Yaskawa INFORM job: DEMO_ROOF_SIDE_0625_3PAINT_41.JBI

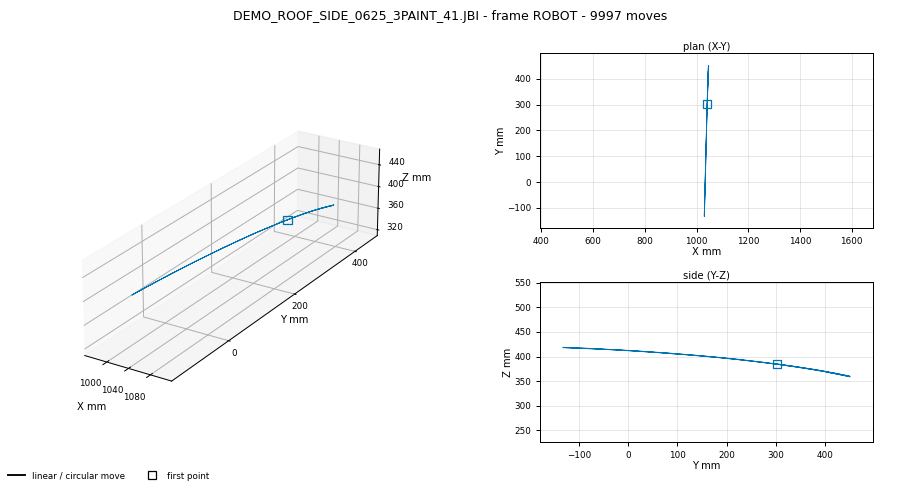
[picture p0: tool path of DEMO_ROOF_SIDE_0625_3PAINT_41.JBI in frame ROBOT, 9997 of 9997 moves have a stored position in this frame; points joined in program order, loops and branches not executed]
/JOB
//NAME DEMO_ROOF_SIDE_0625_3PAINT41
//POS
///NPOS 9997,0,0,0,0,0
///TOOL 0
///USER 0
///POSTYPE ROBOT
///RECTAN
///RCONF 1,0,0,0,0,0,0,0,0,0,0,0,0,0,0,0,0,0,0,0,0,0,0,0
C00000=1041.945,303.509,384.970,171.969,41.641,157.984
C00001=1041.951,303.756,384.937,171.973,41.643,157.985
C00002=1041.958,304.004,384.903,171.977,41.645,157.986
C00003=1041.965,304.251,384.871,171.981,41.648,157.987
C00004=1041.972,304.500,384.838,171.985,41.651,157.987
C00005=1041.979,304.747,384.804,171.988,41.653,157.988
C00006=1041.988,305.081,384.760,171.994,41.656,157.989
C00007=1041.997,305.416,384.715,171.999,41.659,157.990
C00008=1042.007,305.750,384.670,172.004,41.662,157.991
C00009=1042.016,306.084,384.626,172.010,41.665,157.992
C00010=1042.023,306.332,384.592,172.014,41.668,157.993
C00011=1042.030,306.580,384.559,172.018,41.670,157.994
C00012=1042.037,306.827,384.525,172.022,41.672,157.994
C00013=1042.044,307.075,384.491,172.026,41.675,157.995
C00014=1042.050,307.322,384.459,172.030,41.677,157.996
C00015=1042.057,307.570,384.425,172.034,41.680,157.997
C00016=1042.065,307.818,384.392,172.037,41.682,157.998
C00017=1042.072,308.065,384.359,172.041,41.685,157.998
C00018=1042.079,308.313,384.325,172.045,41.687,157.999
C00019=1042.086,308.561,384.292,172.049,41.689,158.000
C00020=1042.092,308.808,384.258,172.053,41.692,158.001
C00021=1042.100,309.056,384.225,172.057,41.694,158.001
C00022=1042.107,309.304,384.192,172.061,41.696,158.002
C00023=1042.114,309.551,384.159,172.065,41.699,158.003
C00024=1042.121,309.798,384.125,172.069,41.702,158.004
C00025=1042.128,310.046,384.091,172.073,41.703,158.005
C00026=1042.135,310.294,384.058,172.077,41.706,158.005
C00027=1042.142,310.541,384.024,172.081,41.709,158.006
C00028=1042.149,310.789,383.991,172.085,41.711,158.007
C00029=1042.156,311.037,383.957,172.089,41.713,158.008
C00030=1042.163,311.284,383.923,172.093,41.716,158.009
C00031=1042.170,311.531,383.890,172.097,41.718,158.009
C00032=1042.178,311.779,383.857,172.101,41.721,158.010
C00033=1042.185,312.027,383.823,172.106,41.723,158.011
C00034=1042.192,312.275,383.789,172.110,41.725,158.012
C00035=1042.198,312.523,383.755,172.114,41.728,158.013
C00036=1042.205,312.770,383.722,172.118,41.730,158.013
C00037=1042.212,313.017,383.688,172.122,41.733,158.014
C00038=1042.219,313.265,383.653,172.125,41.736,158.015
C00039=1042.226,313.512,383.619,172.130,41.739,158.016
C00040=1042.232,313.760,383.585,172.134,41.741,158.017
C00041=1042.239,314.007,383.551,172.138,41.744,158.018
C00042=1042.246,314.255,383.516,172.142,41.746,158.018
C00043=1042.253,314.503,383.483,172.146,41.749,158.019
C00044=1042.259,314.750,383.449,172.150,41.752,158.020
C00045=1042.266,314.997,383.414,172.154,41.754,158.021
C00046=1042.273,315.245,383.380,172.158,41.757,158.022
C00047=1042.280,315.493,383.346,172.162,41.759,158.023
C00048=1042.286,315.741,383.311,172.166,41.762,158.024
C00049=1042.294,315.988,383.277,172.170,41.765,158.024
C00050=1042.300,316.235,383.243,172.175,41.767,158.025
C00051=1042.307,316.483,383.209,172.179,41.770,158.026
C00052=1042.314,316.730,383.174,172.183,41.773,158.027
C00053=1042.321,316.978,383.140,172.187,41.775,158.028
C00054=1042.328,317.226,383.106,172.191,41.778,158.029
C00055=1042.335,317.473,383.071,172.195,41.781,158.029
C00056=1042.342,317.721,383.037,172.200,41.783,158.030
C00057=1042.349,317.968,383.002,172.204,41.786,158.031
C00058=1042.356,318.216,382.968,172.208,41.789,158.032
C00059=1042.362,318.463,382.934,172.212,41.792,158.033
C00060=1042.369,318.710,382.900,172.216,41.794,158.034
C00061=1042.376,318.958,382.865,172.221,41.797,158.035
C00062=1042.386,319.297,382.818,172.227,41.800,158.036
C00063=1042.395,319.636,382.771,172.232,41.804,158.037
C00064=1042.405,319.975,382.724,172.239,41.808,158.038
C00065=1042.415,320.314,382.676,172.244,41.811,158.039
C00066=1042.422,320.562,382.641,172.249,41.814,158.040
C00067=1042.429,320.809,382.607,172.253,41.817,158.041
C00068=1042.435,321.057,382.572,172.257,41.820,158.042
C00069=1042.443,321.304,382.538,172.261,41.822,158.043
C00070=1042.450,321.551,382.502,172.266,41.825,158.044
C00071=1042.457,321.799,382.469,172.270,41.828,158.045
C00072=1042.464,322.046,382.433,172.274,41.831,158.046
C00073=1042.470,322.294,382.398,172.278,41.833,158.047
C00074=1042.478,322.541,382.365,172.283,41.836,158.047
C00075=1042.485,322.789,382.329,172.287,41.839,158.048
C00076=1042.493,323.036,382.294,172.291,41.841,158.049
C00077=1042.499,323.284,382.259,172.296,41.844,158.050
C00078=1042.507,323.531,382.226,172.300,41.847,158.051
C00079=1042.513,323.779,382.190,172.304,41.850,158.052
C00080=1042.521,324.026,382.156,172.310,41.853,158.053
C00081=1042.528,324.273,382.121,172.313,41.855,158.054
C00082=1042.535,324.521,382.085,172.318,41.858,158.055
C00083=1042.542,324.768,382.051,172.323,41.861,158.056
C00084=1042.549,325.016,382.016,172.327,41.864,158.057
C00085=1042.556,325.263,381.982,172.331,41.866,158.057
C00086=1042.564,325.511,381.946,172.336,41.869,158.058
C00087=1042.571,325.759,381.912,172.340,41.872,158.059
C00088=1042.578,326.006,381.877,172.344,41.875,158.060
C00089=1042.585,326.253,381.841,172.349,41.877,158.061
C00090=1042.593,326.501,381.807,172.353,41.881,158.062
C00091=1042.600,326.748,381.771,172.357,41.883,158.063
C00092=1042.607,326.995,381.737,172.362,41.886,158.064
C00093=1042.615,327.244,381.701,172.366,41.889,158.065
C00094=1042.621,327.491,381.666,172.371,41.892,158.066
C00095=1042.629,327.738,381.632,172.375,41.894,158.067
C00096=1042.636,327.986,381.596,172.380,41.897,158.068
C00097=1042.644,328.233,381.562,172.385,41.900,158.069
C00098=1042.651,328.480,381.526,172.389,41.903,158.069
C00099=1042.658,328.728,381.490,172.394,41.906,158.070
C00100=1042.666,328.975,381.456,172.398,41.909,158.071
C00101=1042.672,329.222,381.421,172.402,41.911,158.072
C00102=1042.680,329.470,381.385,172.407,41.914,158.073
C00103=1042.687,329.717,381.349,172.411,41.918,158.074
C00104=1042.694,329.964,381.314,172.417,41.921,158.075
C00105=1042.701,330.213,381.279,172.421,41.924,158.076
C00106=1042.708,330.459,381.243,172.426,41.926,158.077
C00107=1042.715,330.707,381.208,172.430,41.929,158.078
C00108=1042.722,330.955,381.172,172.434,41.932,158.079
C00109=1042.729,331.201,381.136,172.439,41.935,158.080
C00110=1042.737,331.449,381.101,172.443,41.938,158.081
C00111=1042.744,331.696,381.065,172.449,41.941,158.082
C00112=1042.751,331.944,381.030,172.453,41.945,158.083
C00113=1042.758,332.191,380.994,172.458,41.948,158.084
C00114=1042.765,332.438,380.958,172.462,41.951,158.085
C00115=1042.773,332.686,380.922,172.467,41.954,158.086
C00116=1042.779,332.933,380.887,172.471,41.957,158.087
C00117=1042.787,333.181,380.851,172.476,41.960,158.088
C00118=1042.797,333.514,380.803,172.482,41.964,158.089
C00119=1042.807,333.849,380.754,172.489,41.968,158.091
C00120=1042.816,334.183,380.706,172.495,41.972,158.092
C00121=1042.826,334.517,380.658,172.501,41.976,158.093
C00122=1042.833,334.765,380.622,172.506,41.979,158.094
C00123=1042.841,335.012,380.586,172.510,41.982,158.095
C00124=1042.848,335.259,380.550,172.515,41.985,158.096
C00125=1042.856,335.507,380.515,172.520,41.988,158.097
C00126=1042.862,335.754,380.478,172.525,41.992,158.099
C00127=1042.870,336.001,380.442,172.529,41.995,158.100
C00128=1042.877,336.248,380.406,172.534,41.998,158.101
C00129=1042.884,336.496,380.369,172.540,42.001,158.102
C00130=1042.891,336.743,380.333,172.544,42.004,158.103
C00131=1042.898,336.990,380.297,172.549,42.007,158.104
C00132=1042.906,337.238,380.261,172.553,42.011,158.105
C00133=1042.912,337.485,380.224,172.559,42.014,158.106
C00134=1042.920,337.732,380.188,172.563,42.017,158.107
C00135=1042.928,337.979,380.152,172.568,42.020,158.108
C00136=1042.935,338.226,380.116,172.572,42.023,158.109
C00137=1042.942,338.474,380.079,172.577,42.026,158.110
C00138=1042.949,338.721,380.044,172.583,42.030,158.111
C00139=1042.956,338.968,380.007,172.587,42.033,158.112
C00140=1042.963,339.216,379.970,172.592,42.036,158.113
C00141=1042.970,339.463,379.935,172.597,42.040,158.114
C00142=1042.978,339.710,379.898,172.602,42.042,158.115
C00143=1042.985,339.958,379.862,172.607,42.046,158.116
C00144=1042.993,340.205,379.825,172.611,42.049,158.117
C00145=1043.000,340.451,379.789,172.617,42.053,158.119
C00146=1043.008,340.699,379.753,172.621,42.056,158.120
C00147=1043.015,340.947,379.716,172.626,42.059,158.121
C00148=1043.022,341.194,379.680,172.632,42.062,158.122
C00149=1043.030,341.440,379.643,172.636,42.065,158.123
C00150=1043.037,341.688,379.606,172.641,42.069,158.124
C00151=1043.044,341.935,379.570,172.646,42.072,158.125
C00152=1043.051,342.183,379.533,172.651,42.075,158.126
C00153=1043.059,342.430,379.496,172.656,42.079,158.127
C00154=1043.066,342.677,379.460,172.661,42.082,158.128
C00155=1043.074,342.924,379.423,172.666,42.086,158.129
C00156=1043.081,343.172,379.386,172.671,42.089,158.131
C00157=1043.089,343.418,379.349,172.676,42.092,158.132
C00158=1043.095,343.666,379.312,172.681,42.096,158.133
C00159=1043.103,343.912,379.276,172.686,42.099,158.134
C00160=1043.110,344.160,379.239,172.691,42.102,158.135
C00161=1043.118,344.407,379.202,172.696,42.106,158.136
C00162=1043.125,344.655,379.165,172.701,42.109,158.137
C00163=1043.132,344.902,379.128,172.706,42.112,158.138
C00164=1043.140,345.149,379.091,172.712,42.116,158.140
C00165=1043.147,345.396,379.054,172.716,42.120,158.141
C00166=1043.155,345.643,379.017,172.721,42.123,158.142
C00167=1043.162,345.890,378.979,172.727,42.127,158.143
C00168=1043.168,346.137,378.943,172.732,42.130,158.144
C00169=1043.176,346.384,378.906,172.736,42.133,158.145
C00170=1043.184,346.631,378.869,172.742,42.137,158.146
C00171=1043.191,346.878,378.831,172.747,42.140,158.148
C00172=1043.199,347.125,378.794,172.753,42.144,158.149
C00173=1043.206,347.373,378.757,172.757,42.147,158.150
C00174=1043.216,347.704,378.707,172.764,42.152,158.151
C00175=1043.226,348.034,378.658,172.771,42.157,158.153
C00176=1043.236,348.365,378.607,172.779,42.161,158.155
C00177=1043.246,348.695,378.558,172.785,42.166,158.156
C00178=1043.254,348.942,378.520,172.790,42.170,158.157
C00179=1043.261,349.189,378.483,172.795,42.173,158.159
C00180=1043.269,349.436,378.446,172.801,42.177,158.160
C00181=1043.277,349.683,378.408,172.806,42.180,158.161
C00182=1043.284,349.931,378.370,172.812,42.184,158.162
C00183=1043.291,350.178,378.333,172.817,42.188,158.163
C00184=1043.299,350.425,378.296,172.822,42.191,158.165
C00185=1043.306,350.672,378.258,172.827,42.195,158.166
C00186=1043.314,350.919,378.221,172.832,42.198,158.167
C00187=1043.321,351.166,378.183,172.838,42.202,158.168
C00188=1043.328,351.412,378.145,172.843,42.206,158.169
C00189=1043.336,351.660,378.108,172.849,42.209,158.171
C00190=1043.343,351.907,378.070,172.853,42.213,158.172
C00191=1043.351,352.154,378.031,172.859,42.217,158.173
C00192=1043.358,352.401,377.994,172.864,42.221,158.174
C00193=1043.366,352.648,377.956,172.870,42.224,158.176
C00194=1043.373,352.895,377.918,172.875,42.228,158.177
C00195=1043.381,353.142,377.881,172.881,42.232,158.178
C00196=1043.389,353.389,377.843,172.886,42.235,158.179
C00197=1043.396,353.636,377.805,172.892,42.239,158.181
C00198=1043.404,353.883,377.767,172.897,42.243,158.182
C00199=1043.411,354.130,377.729,172.903,42.247,158.183
C00200=1043.419,354.377,377.691,172.908,42.250,158.184
C00201=1043.427,354.624,377.653,172.913,42.255,158.186
C00202=1043.434,354.871,377.616,172.918,42.258,158.187
C00203=1043.441,355.118,377.577,172.924,42.262,158.188
C00204=1043.449,355.365,377.539,172.929,42.266,158.189
C00205=1043.457,355.612,377.501,172.935,42.270,158.191
C00206=1043.464,355.858,377.463,172.940,42.273,158.192
C00207=1043.472,356.106,377.425,172.946,42.277,158.193
C00208=1043.480,356.353,377.387,172.951,42.281,158.194
C00209=1043.487,356.599,377.349,172.957,42.285,158.196
C00210=1043.495,356.847,377.311,172.963,42.289,158.197
C00211=1043.503,357.094,377.272,172.968,42.292,158.198
C00212=1043.511,357.341,377.234,172.974,42.296,158.200
C00213=1043.518,357.587,377.196,172.979,42.300,158.201
C00214=1043.526,357.834,377.157,172.985,42.304,158.202
C00215=1043.533,358.082,377.119,172.990,42.308,158.204
C00216=1043.541,358.329,377.081,172.996,42.312,158.205
C00217=1043.549,358.576,377.042,173.002,42.316,158.206
C00218=1043.556,358.822,377.004,173.007,42.320,158.208
C00219=1043.564,359.069,376.966,173.013,42.324,158.209
C00220=1043.572,359.316,376.927,173.018,42.328,158.210
C00221=1043.580,359.563,376.889,173.025,42.331,158.212
C00222=1043.587,359.810,376.849,173.031,42.335,158.213
C00223=1043.595,360.057,376.811,173.036,42.340,158.214
C00224=1043.603,360.304,376.773,173.042,42.344,158.216
C00225=1043.610,360.550,376.734,173.048,42.348,158.217
C00226=1043.619,360.797,376.695,173.053,42.352,158.218
C00227=1043.626,361.044,376.656,173.059,42.356,158.220
C00228=1043.634,361.291,376.618,173.065,42.360,158.221
C00229=1043.642,361.538,376.579,173.070,42.364,158.222
C00230=1043.652,361.874,376.526,173.078,42.369,158.224
C00231=1043.663,362.211,376.473,173.087,42.375,158.226
C00232=1043.674,362.547,376.421,173.094,42.380,158.228
C00233=1043.683,362.883,376.367,173.102,42.386,158.230
C00234=1043.692,363.130,376.328,173.108,42.390,158.231
C00235=1043.699,363.377,376.289,173.114,42.394,158.233
C00236=1043.707,363.623,376.250,173.119,42.398,158.234
C00237=1043.715,363.870,376.212,173.125,42.403,158.236
C00238=1043.722,364.117,376.172,173.132,42.407,158.237
C00239=1043.730,364.364,376.133,173.138,42.411,158.238
C00240=1043.738,364.610,376.094,173.143,42.416,158.240
C00241=1043.746,364.857,376.054,173.149,42.420,158.241
C00242=1043.753,365.104,376.015,173.155,42.424,158.243
C00243=1043.761,365.350,375.976,173.162,42.428,158.244
C00244=1043.769,365.598,375.937,173.167,42.432,158.245
C00245=1043.777,365.844,375.898,173.173,42.437,158.247
C00246=1043.785,366.091,375.858,173.179,42.441,158.248
C00247=1043.793,366.337,375.819,173.185,42.445,158.250
C00248=1043.800,366.585,375.779,173.192,42.450,158.251
C00249=1043.809,366.831,375.740,173.197,42.454,158.253
C00250=1043.816,367.078,375.700,173.203,42.458,158.254
C00251=1043.824,367.325,375.660,173.210,42.462,158.256
C00252=1043.832,367.571,375.621,173.216,42.467,158.257
C00253=1043.840,367.818,375.581,173.222,42.471,158.259
C00254=1043.848,368.065,375.543,173.227,42.475,158.260
C00255=1043.856,368.312,375.503,173.234,42.480,158.262
C00256=1043.864,368.559,375.464,173.240,42.484,158.263
C00257=1043.872,368.806,375.424,173.246,42.488,158.265
C00258=1043.880,369.052,375.384,173.252,42.493,158.266
C00259=1043.888,369.299,375.344,173.258,42.497,158.268
C00260=1043.896,369.545,375.305,173.264,42.502,158.269
C00261=1043.903,369.792,375.266,173.271,42.506,158.271
C00262=1043.912,370.038,375.225,173.277,42.510,158.272
C00263=1043.920,370.285,375.186,173.283,42.515,158.274
C00264=1043.928,370.531,375.146,173.290,42.519,158.275
C00265=1043.936,370.778,375.106,173.295,42.524,158.277
C00266=1043.944,371.025,375.066,173.302,42.528,158.278
C00267=1043.952,371.271,375.026,173.308,42.533,158.280
C00268=1043.960,371.518,374.986,173.314,42.537,158.281
C00269=1043.968,371.765,374.947,173.321,42.542,158.283
C00270=1043.976,372.011,374.906,173.327,42.546,158.284
C00271=1043.984,372.258,374.866,173.333,42.551,158.286
C00272=1043.992,372.504,374.825,173.340,42.556,158.288
C00273=1044.000,372.751,374.785,173.346,42.560,158.289
C00274=1044.007,372.998,374.745,173.353,42.565,158.291
C00275=1044.015,373.245,374.705,173.359,42.569,158.292
C00276=1044.024,373.491,374.665,173.366,42.574,158.294
C00277=1044.032,373.737,374.625,173.372,42.579,158.295
C00278=1044.040,373.984,374.584,173.377,42.583,158.297
C00279=1044.048,374.231,374.544,173.384,42.588,158.299
C00280=1044.056,374.478,374.503,173.390,42.593,158.300
C00281=1044.064,374.724,374.463,173.397,42.597,158.302
C00282=1044.072,374.971,374.423,173.403,42.602,158.304
C00283=1044.080,375.217,374.382,173.410,42.607,158.305
C00284=1044.089,375.463,374.342,173.416,42.612,158.307
C00285=1044.097,375.710,374.301,173.423,42.616,158.308
C00286=1044.105,375.944,374.263,173.429,42.621,158.310
C00287=1044.112,376.178,374.225,173.436,42.625,158.311
C00288=1044.121,376.412,374.186,173.442,42.630,158.313
C00289=1044.127,376.646,374.147,173.448,42.634,158.315
C00290=1044.136,376.881,374.108,173.455,42.639,158.316
C00291=1044.143,377.115,374.070,173.461,42.643,158.318
C00292=1044.151,377.349,374.031,173.467,42.648,158.319
C00293=1044.159,377.583,373.993,173.474,42.653,158.321
C00294=1044.172,377.964,373.930,173.484,42.660,158.323
C00295=1044.185,378.344,373.868,173.494,42.668,158.326
C00296=1044.198,378.724,373.804,173.504,42.675,158.329
C00297=1044.211,379.105,373.741,173.515,42.683,158.331
C00298=1044.218,379.352,373.700,173.522,42.687,158.333
C00299=1044.227,379.599,373.659,173.528,42.693,158.335
C00300=1044.235,379.845,373.618,173.535,42.698,158.336
C00301=1044.243,380.091,373.577,173.542,42.702,158.338
C00302=1044.251,380.338,373.535,173.548,42.708,158.340
C00303=1044.259,380.584,373.494,173.555,42.712,158.342
C00304=1044.268,380.831,373.453,173.563,42.717,158.343
C00305=1044.276,381.076,373.412,173.569,42.722,158.345
C00306=1044.284,381.324,373.370,173.576,42.727,158.347
C00307=1044.293,381.569,373.329,173.583,42.733,158.349
C00308=1044.301,381.816,373.288,173.589,42.738,158.350
C00309=1044.310,382.062,373.246,173.597,42.743,158.352
C00310=1044.318,382.309,373.205,173.604,42.748,158.354
C00311=1044.326,382.555,373.164,173.611,42.753,158.356
C00312=1044.335,382.801,373.122,173.617,42.758,158.357
C00313=1044.343,383.048,373.081,173.624,42.763,158.359
C00314=1044.351,383.294,373.039,173.632,42.769,158.361
C00315=1044.359,383.540,372.998,173.639,42.774,158.363
C00316=1044.368,383.787,372.957,173.646,42.779,158.365
C00317=1044.377,384.033,372.915,173.652,42.784,158.366
C00318=1044.384,384.279,372.873,173.660,42.790,158.368
C00319=1044.393,384.526,372.831,173.667,42.794,158.370
C00320=1044.402,384.772,372.789,173.674,42.800,158.372
C00321=1044.410,385.018,372.747,173.681,42.805,158.374
C00322=1044.419,385.264,372.706,173.688,42.810,158.376
C00323=1044.428,385.511,372.664,173.695,42.815,158.377
C00324=1044.436,385.756,372.623,173.702,42.821,158.379
C00325=1044.444,386.003,372.580,173.710,42.826,158.381
C00326=1044.453,386.249,372.539,173.717,42.831,158.383
C00327=1044.462,386.496,372.497,173.724,42.836,158.385
C00328=1044.470,386.742,372.455,173.732,42.842,158.387
C00329=1044.479,386.988,372.413,173.739,42.847,158.389
C00330=1044.488,387.235,372.372,173.747,42.853,158.390
C00331=1044.496,387.481,372.329,173.754,42.858,158.392
C00332=1044.505,387.728,372.288,173.761,42.863,158.394
C00333=1044.514,387.973,372.245,173.767,42.869,158.396
C00334=1044.522,388.220,372.203,173.775,42.874,158.398
C00335=1044.531,388.466,372.161,173.782,42.880,158.400
C00336=1044.540,388.711,372.119,173.790,42.885,158.402
C00337=1044.548,388.958,372.077,173.797,42.890,158.404
C00338=1044.556,389.204,372.034,173.805,42.896,158.406
C00339=1044.565,389.450,371.992,173.812,42.902,158.408
C00340=1044.574,389.697,371.949,173.820,42.907,158.410
C00341=1044.583,389.943,371.907,173.827,42.913,158.411
C00342=1044.596,390.332,371.840,173.839,42.922,158.415
C00343=1044.610,390.722,371.773,173.851,42.930,158.418
C00344=1044.624,391.111,371.706,173.863,42.939,158.421
C00345=1044.638,391.500,371.638,173.875,42.948,158.424
C00346=1044.646,391.746,371.595,173.883,42.954,158.426
C00347=1044.655,391.992,371.552,173.891,42.959,158.428
C00348=1044.664,392.238,371.510,173.898,42.965,158.430
C00349=1044.673,392.484,371.467,173.906,42.971,158.432
C00350=1044.682,392.731,371.423,173.913,42.977,158.434
C00351=1044.690,392.977,371.380,173.921,42.983,158.436
C00352=1044.699,393.223,371.338,173.929,42.988,158.438
C00353=1044.708,393.469,371.295,173.936,42.994,158.440
C00354=1044.716,393.715,371.252,173.945,43.000,158.442
C00355=1044.725,393.961,371.209,173.952,43.006,158.444
C00356=1044.734,394.207,371.167,173.960,43.012,158.447
C00357=1044.743,394.453,371.123,173.968,43.018,158.449
C00358=1044.752,394.699,371.080,173.975,43.023,158.451
C00359=1044.761,394.945,371.036,173.984,43.029,158.453
C00360=1044.770,395.191,370.994,173.992,43.035,158.455
C00361=1044.779,395.437,370.951,173.999,43.041,158.457
C00362=1044.787,395.683,370.907,174.007,43.047,158.459
C00363=1044.796,395.929,370.864,174.016,43.053,158.461
C00364=1044.805,396.176,370.820,174.023,43.059,158.463
C00365=1044.814,396.421,370.777,174.031,43.065,158.465
C00366=1044.823,396.667,370.734,174.040,43.070,158.468
C00367=1044.832,396.913,370.689,174.048,43.077,158.470
C00368=1044.841,397.159,370.647,174.055,43.083,158.472
C00369=1044.850,397.404,370.603,174.063,43.089,158.474
C00370=1044.859,397.651,370.560,174.072,43.095,158.476
C00371=1044.868,397.897,370.516,174.080,43.101,158.478
C00372=1044.877,398.143,370.472,174.089,43.107,158.481
C00373=1044.886,398.389,370.429,174.096,43.113,158.483
C00374=1044.895,398.635,370.385,174.104,43.120,158.485
C00375=1044.904,398.880,370.341,174.113,43.125,158.487
C00376=1044.914,399.126,370.297,174.121,43.132,158.490
C00377=1044.922,399.372,370.253,174.129,43.138,158.492
C00378=1044.932,399.618,370.209,174.137,43.144,158.494
C00379=1044.940,399.864,370.166,174.145,43.151,158.496
C00380=1044.950,400.110,370.122,174.154,43.156,158.498
C00381=1044.959,400.356,370.078,174.162,43.163,158.501
C00382=1044.968,400.602,370.034,174.171,43.169,158.503
C00383=1044.977,400.848,369.990,174.179,43.175,158.505
C00384=1044.987,401.094,369.946,174.188,43.182,158.508
C00385=1044.995,401.339,369.901,174.196,43.188,158.510
C00386=1045.005,401.585,369.857,174.204,43.194,158.512
C00387=1045.014,401.831,369.813,174.212,43.201,158.514
C00388=1045.023,402.077,369.769,174.221,43.207,158.517
C00389=1045.032,402.323,369.725,174.229,43.213,158.519
C00390=1045.042,402.569,369.680,174.238,43.220,158.521
C00391=1045.051,402.815,369.635,174.247,43.227,158.524
C00392=1045.060,403.060,369.591,174.255,43.233,158.526
C00393=1045.069,403.306,369.547,174.264,43.239,158.528
C00394=1045.078,403.552,369.503,174.272,43.246,158.531
C00395=1045.087,403.798,369.457,174.281,43.252,158.533
C00396=1045.097,404.044,369.413,174.290,43.259,158.535
C00397=1045.107,404.290,369.368,174.299,43.266,158.538
C00398=1045.122,404.698,369.294,174.314,43.277,158.542
C00399=1045.137,405.106,369.220,174.328,43.287,158.546
C00400=1045.152,405.515,369.145,174.343,43.299,158.550
C00401=1045.168,405.923,369.070,174.357,43.310,158.554
C00402=1045.178,406.169,369.025,174.367,43.317,158.557
C00403=1045.187,406.415,368.980,174.376,43.323,158.559
C00404=1045.196,406.660,368.935,174.384,43.330,158.562
C00405=1045.205,406.906,368.890,174.393,43.337,158.564
C00406=1045.215,407.152,368.845,174.402,43.344,158.566
C00407=1045.224,407.397,368.799,174.412,43.351,158.569
C00408=1045.234,407.643,368.755,174.421,43.357,158.571
C00409=1045.243,407.889,368.709,174.429,43.364,158.574
C00410=1045.253,408.135,368.664,174.438,43.371,158.576
C00411=1045.262,408.381,368.619,174.447,43.378,158.579
C00412=1045.272,408.626,368.573,174.457,43.385,158.582
C00413=1045.282,408.871,368.528,174.466,43.392,158.584
C00414=1045.291,409.118,368.482,174.475,43.398,158.587
C00415=1045.301,409.363,368.437,174.485,43.406,158.589
C00416=1045.310,409.608,368.391,174.494,43.412,158.592
C00417=1045.320,409.854,368.347,174.503,43.420,158.594
C00418=1045.330,410.100,368.300,174.513,43.426,158.597
C00419=1045.340,410.345,368.255,174.522,43.434,158.600
C00420=1045.349,410.591,368.209,174.531,43.440,158.602
C00421=1045.359,410.837,368.164,174.541,43.448,158.605
C00422=1045.368,411.082,368.118,174.550,43.455,158.608
C00423=1045.379,411.328,368.073,174.560,43.462,158.610
C00424=1045.388,411.573,368.026,174.569,43.469,158.613
C00425=1045.399,411.819,367.981,174.579,43.476,158.615
C00426=1045.408,412.065,367.935,174.588,43.483,158.618
C00427=1045.418,412.311,367.889,174.598,43.491,158.621
C00428=1045.428,412.556,367.843,174.607,43.498,158.623
C00429=1045.437,412.802,367.797,174.617,43.505,158.626
C00430=1045.447,413.047,367.750,174.627,43.512,158.629
C00431=1045.457,413.293,367.704,174.637,43.519,158.632
C00432=1045.467,413.538,367.658,174.646,43.527,158.634
C00433=1045.477,413.783,367.612,174.656,43.534,158.637
C00434=1045.486,414.029,367.565,174.665,43.542,158.640
C00435=1045.496,414.275,367.519,174.676,43.549,158.643
C00436=1045.506,414.520,367.472,174.686,43.556,158.645
C00437=1045.516,414.766,367.426,174.695,43.564,158.648
C00438=1045.526,415.011,367.380,174.705,43.571,158.651
C00439=1045.536,415.257,367.334,174.716,43.579,158.654
C00440=1045.546,415.502,367.286,174.725,43.587,158.657
C00441=1045.556,415.748,367.240,174.735,43.594,158.659
C00442=1045.566,415.993,367.193,174.746,43.601,158.662
C00443=1045.575,416.238,367.146,174.755,43.609,158.665
C00444=1045.585,416.484,367.099,174.765,43.617,158.668
C00445=1045.596,416.729,367.053,174.776,43.624,158.671
C00446=1045.606,416.974,367.006,174.786,43.632,158.674
C00447=1045.616,417.220,366.960,174.797,43.640,158.677
C00448=1045.626,417.466,366.912,174.806,43.647,158.680
C00449=1045.636,417.711,366.865,174.817,43.655,158.683
C00450=1045.647,417.956,366.818,174.827,43.663,158.685
C00451=1045.657,418.202,366.771,174.838,43.670,158.688
C00452=1045.667,418.447,366.724,174.848,43.678,158.691
C00453=1045.677,418.693,366.677,174.859,43.686,158.694
C00454=1045.686,418.901,366.637,174.867,43.693,158.697
C00455=1045.695,419.108,366.597,174.876,43.699,158.699
C00456=1045.703,419.317,366.557,174.885,43.706,158.702
C00457=1045.712,419.525,366.517,174.894,43.713,158.705
C00458=1045.720,419.733,366.476,174.902,43.719,158.707
C00459=1045.729,419.941,366.436,174.912,43.726,158.710
C00460=1045.738,420.149,366.396,174.921,43.732,158.712
C00461=1045.747,420.357,366.356,174.929,43.739,158.715
C00462=1045.757,420.602,366.309,174.940,43.747,158.718
C00463=1045.767,420.847,366.260,174.951,43.755,158.721
C00464=1045.777,421.092,366.213,174.961,43.763,158.724
C00465=1045.787,421.338,366.166,174.973,43.771,158.727
C00466=1045.798,421.583,366.117,174.984,43.779,158.730
C00467=1045.808,421.828,366.070,174.995,43.787,158.733
C00468=1045.819,422.073,366.022,175.005,43.796,158.736
C00469=1045.829,422.318,365.974,175.016,43.804,158.740
C00470=1045.839,422.564,365.926,175.027,43.812,158.743
C00471=1045.850,422.809,365.878,175.038,43.820,158.746
C00472=1045.861,423.054,365.830,175.049,43.828,158.749
C00473=1045.871,423.299,365.783,175.061,43.837,158.752
C00474=1045.882,423.544,365.735,175.072,43.845,158.755
C00475=1045.892,423.790,365.686,175.082,43.853,158.759
C00476=1045.902,424.034,365.638,175.093,43.862,158.762
C00477=1045.914,424.280,365.590,175.105,43.870,158.765
C00478=1045.924,424.524,365.542,175.116,43.878,158.768
C00479=1045.935,424.770,365.493,175.127,43.887,158.772
C00480=1045.946,425.015,365.444,175.139,43.895,158.775
C00481=1045.956,425.260,365.397,175.150,43.904,158.778
C00482=1045.967,425.505,365.348,175.161,43.912,158.781
C00483=1045.977,425.750,365.300,175.174,43.921,158.785
C00484=1045.988,425.995,365.251,175.185,43.929,158.788
C00485=1045.998,426.240,365.202,175.197,43.937,158.791
C00486=1046.009,426.485,365.153,175.208,43.946,158.795
C00487=1046.020,426.730,365.104,175.220,43.955,158.798
C00488=1046.031,426.976,365.056,175.231,43.963,158.802
C00489=1046.042,427.220,365.007,175.243,43.972,158.805
C00490=1046.052,427.465,364.958,175.255,43.981,158.808
C00491=1046.063,427.710,364.909,175.267,43.990,158.812
C00492=1046.074,427.955,364.860,175.278,43.998,158.815
C00493=1046.085,428.199,364.811,175.290,44.007,158.819
C00494=1046.095,428.445,364.762,175.302,44.016,158.822
C00495=1046.107,428.690,364.713,175.314,44.025,158.826
C00496=1046.118,428.934,364.664,175.326,44.033,158.829
C00497=1046.129,429.179,364.615,175.338,44.042,158.833
C00498=1046.139,429.425,364.565,175.350,44.051,158.836
C00499=1046.151,429.669,364.516,175.363,44.060,158.840
C00500=1046.162,429.914,364.466,175.375,44.069,158.843
C00501=1046.172,430.159,364.417,175.386,44.078,158.847
C00502=1046.184,430.404,364.367,175.399,44.087,158.850
C00503=1046.195,430.649,364.317,175.411,44.096,158.854
C00504=1046.205,430.894,364.268,175.424,44.105,158.858
C00505=1046.216,431.138,364.218,175.436,44.114,158.861
C00506=1046.228,431.383,364.169,175.448,44.123,158.865
C00507=1046.238,431.628,364.119,175.461,44.132,158.868
C00508=1046.250,431.873,364.068,175.473,44.141,158.872
C00509=1046.262,432.117,364.018,175.486,44.151,158.876
C00510=1046.272,432.362,363.969,175.499,44.160,158.880
C00511=1046.283,432.607,363.919,175.511,44.169,158.883
C00512=1046.295,432.851,363.869,175.524,44.178,158.887
C00513=1046.306,433.096,363.819,175.537,44.188,158.891
C00514=1046.316,433.315,363.774,175.549,44.196,158.894
C00515=1046.326,433.534,363.729,175.560,44.204,158.897
C00516=1046.337,433.754,363.684,175.572,44.213,158.901
C00517=1046.346,433.973,363.639,175.583,44.221,158.904
C00518=1046.357,434.192,363.594,175.595,44.230,158.908
C00519=1046.367,434.412,363.548,175.606,44.238,158.911
C00520=1046.378,434.630,363.504,175.618,44.247,158.915
C00521=1046.388,434.850,363.458,175.630,44.255,158.918
C00522=1046.399,435.094,363.408,175.643,44.265,158.922
C00523=1046.411,435.339,363.358,175.656,44.274,158.926
C00524=1046.423,435.584,363.306,175.669,44.283,158.930
C00525=1046.435,435.828,363.257,175.683,44.293,158.934
C00526=1046.446,436.073,363.206,175.696,44.303,158.937
C00527=1046.457,436.317,363.155,175.709,44.312,158.941
C00528=1046.469,436.562,363.104,175.723,44.323,158.946
C00529=1046.481,436.806,363.053,175.736,44.332,158.949
C00530=1046.492,437.050,363.002,175.749,44.342,158.953
C00531=1046.504,437.295,362.951,175.764,44.352,158.958
C00532=1046.516,437.540,362.900,175.777,44.361,158.961
C00533=1046.527,437.784,362.848,175.791,44.371,158.966
C00534=1046.539,438.028,362.797,175.804,44.381,158.970
C00535=1046.551,438.272,362.746,175.819,44.391,158.974
C00536=1046.562,438.517,362.694,175.832,44.401,158.978
C00537=1046.574,438.762,362.643,175.846,44.411,158.982
C00538=1046.586,439.006,362.591,175.860,44.421,158.986
C00539=1046.598,439.251,362.540,175.874,44.431,158.990
C00540=1046.610,439.495,362.489,175.888,44.441,158.994
C00541=1046.622,439.739,362.437,175.903,44.451,158.999
C00542=1046.634,439.983,362.385,175.916,44.462,159.003
C00543=1046.646,440.228,362.334,175.931,44.472,159.007
C00544=1046.658,440.472,362.282,175.945,44.482,159.011
C00545=1046.670,440.716,362.230,175.960,44.492,159.016
C00546=1046.682,440.960,362.178,175.974,44.503,159.020
C00547=1046.694,441.204,362.126,175.988,44.513,159.024
C00548=1046.706,441.449,362.075,176.003,44.523,159.029
C00549=1046.718,441.693,362.022,176.017,44.533,159.033
C00550=1046.731,441.937,361.969,176.032,44.544,159.037
C00551=1046.743,442.181,361.917,176.047,44.554,159.042
C00552=1046.755,442.425,361.865,176.062,44.565,159.046
C00553=1046.767,442.669,361.813,176.076,44.575,159.051
C00554=1046.779,442.914,361.760,176.091,44.586,159.055
C00555=1046.791,443.158,361.708,176.106,44.596,159.059
C00556=1046.804,443.402,361.656,176.121,44.607,159.064
C00557=1046.816,443.646,361.603,176.137,44.617,159.068
C00558=1046.829,443.890,361.550,176.152,44.628,159.073
C00559=1046.841,444.135,361.497,176.167,44.638,159.077
C00560=1046.853,444.378,361.445,176.182,44.649,159.082
C00561=1046.866,444.622,361.392,176.197,44.660,159.087
C00562=1046.879,444.866,361.339,176.213,44.671,159.091
C00563=1046.891,445.110,361.287,176.228,44.681,159.096
C00564=1046.904,445.354,361.234,176.243,44.693,159.101
C00565=1046.917,445.597,361.181,176.259,44.703,159.105
C00566=1046.930,445.840,361.129,176.275,44.714,159.110
C00567=1046.943,446.083,361.076,176.290,44.725,159.114
C00568=1046.958,446.327,361.025,176.306,44.735,159.119
C00569=1046.973,446.571,360.974,176.322,44.745,159.123
C00570=1046.989,446.815,360.924,176.338,44.756,159.128
C00571=1047.006,447.058,360.874,176.354,44.766,159.132
C00572=1047.022,447.302,360.825,176.370,44.775,159.137
C00573=1047.040,447.547,360.776,176.386,44.785,159.141
C00574=1047.066,447.882,360.710,176.408,44.798,159.147
C00575=1047.093,448.217,360.645,176.430,44.811,159.153
C00576=1047.121,448.552,360.581,176.453,44.824,159.159
C00577=1047.150,448.888,360.517,176.475,44.837,159.165
C00578=1047.172,449.133,360.472,176.492,44.845,159.169
C00579=1047.195,449.377,360.427,176.509,44.854,159.174
C00580=1047.218,449.623,360.382,176.526,44.863,159.178
C00581=1047.242,449.868,360.338,176.543,44.871,159.182
C00582=1047.267,450.113,360.294,176.560,44.880,159.186
C00583=1047.292,450.359,360.252,176.576,44.888,159.190
C00584=1047.318,450.604,360.209,176.594,44.896,159.195
C00585=1047.345,450.849,360.168,176.611,44.905,159.199
C00586=1047.037,450.883,359.861,176.612,44.991,159.224
C00587=1047.011,450.638,359.903,176.595,44.983,159.220
C00588=1046.984,450.392,359.945,176.578,44.975,159.216
C00589=1046.958,450.147,359.988,176.561,44.967,159.212
C00590=1046.933,449.901,360.032,176.544,44.958,159.208
C00591=1046.909,449.656,360.076,176.526,44.950,159.204
C00592=1046.886,449.411,360.120,176.510,44.941,159.199
C00593=1046.863,449.166,360.165,176.493,44.933,159.195
C00594=1046.840,448.921,360.211,176.476,44.924,159.191
C00595=1046.812,448.603,360.270,176.455,44.912,159.185
C00596=1046.785,448.284,360.331,176.433,44.900,159.180
C00597=1046.760,447.966,360.392,176.411,44.888,159.174
C00598=1046.735,447.649,360.455,176.390,44.876,159.168
C00599=1046.717,447.405,360.503,176.374,44.866,159.164
C00600=1046.699,447.161,360.553,176.358,44.856,159.159
C00601=1046.682,446.916,360.602,176.342,44.846,159.155
C00602=1046.666,446.673,360.652,176.326,44.836,159.150
C00603=1046.650,446.429,360.703,176.310,44.827,159.146
C00604=1046.636,446.185,360.754,176.294,44.816,159.141
C00605=1046.621,445.942,360.806,176.278,44.805,159.137
C00606=1046.607,445.699,360.858,176.263,44.795,159.132
C00607=1046.595,445.456,360.911,176.247,44.784,159.127
C00608=1046.582,445.212,360.963,176.231,44.774,159.123
C00609=1046.570,444.968,361.016,176.216,44.763,159.118
C00610=1046.557,444.725,361.069,176.201,44.752,159.113
C00611=1046.545,444.481,361.122,176.185,44.741,159.109
C00612=1046.532,444.237,361.174,176.170,44.731,159.104
C00613=1046.519,443.993,361.227,176.155,44.720,159.100
C00614=1046.507,443.748,361.280,176.140,44.710,159.095
C00615=1046.495,443.505,361.332,176.125,44.699,159.091
C00616=1046.482,443.261,361.385,176.109,44.689,159.086
C00617=1046.470,443.017,361.437,176.094,44.678,159.082
C00618=1046.457,442.772,361.490,176.079,44.668,159.077
C00619=1046.445,442.528,361.543,176.064,44.657,159.073
C00620=1046.433,442.284,361.595,176.049,44.647,159.068
C00621=1046.421,442.040,361.647,176.034,44.637,159.064
C00622=1046.408,441.796,361.699,176.020,44.626,159.060
C00623=1046.396,441.552,361.751,176.005,44.616,159.055
C00624=1046.384,441.307,361.803,175.990,44.606,159.051
C00625=1046.373,441.063,361.856,175.976,44.596,159.047
C00626=1046.360,440.818,361.908,175.961,44.585,159.042
C00627=1046.348,440.574,361.960,175.947,44.575,159.038
C00628=1046.336,440.330,362.012,175.933,44.565,159.034
C00629=1046.324,440.085,362.063,175.918,44.555,159.030
C00630=1046.312,439.842,362.115,175.904,44.544,159.025
C00631=1046.300,439.597,362.167,175.890,44.535,159.021
C00632=1046.288,439.353,362.218,175.876,44.524,159.017
C00633=1046.276,439.109,362.270,175.861,44.515,159.013
C00634=1046.264,438.864,362.321,175.848,44.505,159.009
C00635=1046.252,438.620,362.373,175.833,44.495,159.004
C00636=1046.241,438.376,362.424,175.819,44.485,159.000
C00637=1046.229,438.131,362.475,175.806,44.475,158.996
C00638=1046.217,437.887,362.527,175.791,44.465,158.992
C00639=1046.205,437.642,362.578,175.778,44.456,158.988
C00640=1046.193,437.398,362.630,175.764,44.445,158.984
C00641=1046.182,437.153,362.680,175.751,44.436,158.980
C00642=1046.170,436.909,362.731,175.737,44.426,158.976
C00643=1046.159,436.664,362.783,175.723,44.416,158.972
C00644=1046.146,436.420,362.833,175.709,44.407,158.968
C00645=1046.135,436.176,362.884,175.696,44.397,158.964
C00646=1046.123,435.931,362.935,175.683,44.387,158.960
C00647=1046.112,435.686,362.986,175.669,44.378,158.956
C00648=1046.101,435.442,363.036,175.656,44.368,158.952
C00649=1046.089,435.197,363.087,175.643,44.359,158.948
C00650=1046.076,434.952,363.138,175.630,44.349,158.944
C00651=1046.067,434.732,363.183,175.618,44.341,158.941
C00652=1046.056,434.512,363.229,175.605,44.333,158.937
C00653=1046.046,434.292,363.274,175.594,44.324,158.934
C00654=1046.036,434.072,363.320,175.582,44.316,158.930
C00655=1046.025,433.852,363.364,175.570,44.307,158.927
C00656=1046.015,433.632,363.409,175.559,44.299,158.924
C00657=1046.005,433.411,363.455,175.547,44.291,158.920
C00658=1045.995,433.191,363.500,175.536,44.282,158.917
C00659=1045.982,432.946,363.550,175.523,44.273,158.913
C00660=1045.972,432.702,363.600,175.510,44.264,158.909
C00661=1045.961,432.457,363.650,175.498,44.255,158.906
C00662=1045.950,432.213,363.700,175.485,44.245,158.902
C00663=1045.938,431.968,363.750,175.472,44.236,158.898
C00664=1045.927,431.723,363.800,175.460,44.227,158.895
C00665=1045.916,431.478,363.850,175.447,44.218,158.891
C00666=1045.905,431.234,363.899,175.434,44.209,158.887
C00667=1045.894,430.989,363.949,175.422,44.200,158.884
C00668=1045.883,430.744,363.999,175.409,44.191,158.880
C00669=1045.871,430.499,364.048,175.397,44.182,158.876
C00670=1045.860,430.255,364.098,175.385,44.173,158.873
C00671=1045.850,430.010,364.148,175.373,44.164,158.869
C00672=1045.838,429.765,364.197,175.360,44.155,158.866
C00673=1045.828,429.520,364.247,175.348,44.146,158.862
C00674=1045.817,429.275,364.296,175.335,44.138,158.859
C00675=1045.806,429.030,364.345,175.324,44.129,158.855
C00676=1045.795,428.785,364.395,175.312,44.120,158.852
C00677=1045.784,428.540,364.444,175.299,44.111,158.848
C00678=1045.773,428.295,364.493,175.288,44.103,158.845
C00679=1045.762,428.051,364.542,175.275,44.094,158.841
C00680=1045.751,427.805,364.591,175.263,44.085,158.838
C00681=1045.740,427.560,364.640,175.252,44.076,158.834
C00682=1045.728,427.315,364.689,175.240,44.067,158.831
C00683=1045.719,427.071,364.738,175.228,44.059,158.827
C00684=1045.707,426.826,364.787,175.216,44.051,158.824
C00685=1045.697,426.580,364.836,175.205,44.042,158.821
C00686=1045.686,426.336,364.884,175.193,44.033,158.817
C00687=1045.675,426.091,364.933,175.182,44.025,158.814
C00688=1045.664,425.846,364.982,175.169,44.017,158.811
C00689=1045.654,425.601,365.030,175.158,44.008,158.807
C00690=1045.643,425.355,365.079,175.147,44.000,158.804
C00691=1045.632,425.110,365.127,175.135,43.991,158.801
C00692=1045.622,424.866,365.176,175.124,43.983,158.797
C00693=1045.611,424.620,365.225,175.112,43.974,158.794
C00694=1045.601,424.376,365.273,175.101,43.966,158.791
C00695=1045.590,424.130,365.321,175.090,43.958,158.788
C00696=1045.579,423.886,365.369,175.078,43.949,158.784
C00697=1045.568,423.640,365.417,175.067,43.941,158.781
C00698=1045.559,423.395,365.465,175.056,43.933,158.778
C00699=1045.547,423.149,365.514,175.045,43.925,158.775
C00700=1045.537,422.905,365.561,175.034,43.917,158.772
C00701=1045.526,422.659,365.610,175.022,43.909,158.768
C00702=1045.516,422.414,365.657,175.012,43.900,158.765
C00703=1045.505,422.169,365.705,175.001,43.892,158.762
C00704=1045.494,421.924,365.753,174.990,43.884,158.759
C00705=1045.485,421.678,365.801,174.979,43.876,158.756
C00706=1045.474,421.434,365.849,174.968,43.868,158.753
C00707=1045.464,421.188,365.896,174.958,43.860,158.750
C00708=1045.453,420.942,365.944,174.946,43.852,158.746
C00709=1045.443,420.698,365.992,174.935,43.844,158.743
C00710=1045.432,420.452,366.039,174.925,43.837,158.740
C00711=1045.424,420.243,366.080,174.916,43.829,158.738
C00712=1045.415,420.034,366.120,174.907,43.823,158.735
C00713=1045.406,419.825,366.161,174.897,43.816,158.733
C00714=1045.398,419.616,366.201,174.889,43.810,158.730
C00715=1045.389,419.407,366.241,174.879,43.803,158.727
C00716=1045.380,419.198,366.282,174.870,43.797,158.725
C00717=1045.372,418.989,366.322,174.862,43.790,158.722
C00718=1045.363,418.780,366.362,174.852,43.783,158.720
C00719=1045.353,418.534,366.410,174.842,43.775,158.717
C00720=1045.342,418.289,366.457,174.831,43.767,158.714
C00721=1045.332,418.044,366.504,174.821,43.760,158.711
C00722=1045.322,417.798,366.551,174.811,43.752,158.708
C00723=1045.312,417.553,366.598,174.800,43.745,158.705
C00724=1045.302,417.307,366.645,174.790,43.737,158.702
C00725=1045.292,417.062,366.692,174.779,43.730,158.699
C00726=1045.281,416.817,366.739,174.770,43.722,158.696
C00727=1045.272,416.571,366.786,174.760,43.714,158.693
C00728=1045.261,416.326,366.832,174.749,43.707,158.691
C00729=1045.251,416.081,366.878,174.739,43.699,158.688
C00730=1045.241,415.835,366.926,174.729,43.692,158.685
C00731=1045.231,415.589,366.972,174.719,43.684,158.682
C00732=1045.221,415.344,367.019,174.709,43.676,158.679
C00733=1045.211,415.098,367.066,174.698,43.669,158.676
C00734=1045.201,414.853,367.111,174.689,43.662,158.674
C00735=1045.191,414.608,367.159,174.679,43.654,158.671
C00736=1045.181,414.362,367.205,174.668,43.647,158.668
C00737=1045.172,414.117,367.251,174.659,43.640,158.665
C00738=1045.162,413.871,367.298,174.649,43.632,158.662
C00739=1045.151,413.625,367.344,174.640,43.625,158.660
C00740=1045.142,413.381,367.391,174.630,43.617,158.657
C00741=1045.132,413.135,367.437,174.619,43.610,158.654
C00742=1045.123,412.890,367.483,174.610,43.603,158.651
C00743=1045.113,412.644,367.530,174.600,43.596,158.649
C00744=1045.103,412.399,367.576,174.591,43.589,158.646
C00745=1045.093,412.152,367.621,174.581,43.582,158.643
C00746=1045.083,411.906,367.668,174.572,43.574,158.641
C00747=1045.073,411.662,367.713,174.561,43.567,158.638
C00748=1045.064,411.415,367.759,174.552,43.561,158.635
C00749=1045.054,411.170,367.804,174.542,43.553,158.633
C00750=1045.044,410.924,367.851,174.533,43.546,158.630
C00751=1045.034,410.679,367.896,174.524,43.539,158.627
C00752=1045.025,410.434,367.942,174.514,43.532,158.625
C00753=1045.014,410.187,367.987,174.505,43.526,158.622
C00754=1045.005,409.942,368.033,174.495,43.518,158.620
C00755=1044.995,409.696,368.078,174.486,43.512,158.617
C00756=1044.986,409.451,368.125,174.477,43.504,158.614
C00757=1044.976,409.205,368.169,174.467,43.498,158.612
C00758=1044.966,408.959,368.215,174.458,43.491,158.609
C00759=1044.956,408.714,368.261,174.448,43.484,158.607
C00760=1044.946,408.468,368.305,174.439,43.477,158.604
C00761=1044.937,408.222,368.351,174.430,43.470,158.602
C00762=1044.928,407.977,368.396,174.421,43.463,158.599
C00763=1044.918,407.730,368.442,174.411,43.457,158.597
C00764=1044.908,407.485,368.487,174.403,43.450,158.594
C00765=1044.899,407.240,368.532,174.394,43.443,158.592
C00766=1044.889,406.994,368.577,174.385,43.436,158.589
C00767=1044.881,406.748,368.623,174.376,43.430,158.587
C00768=1044.871,406.503,368.668,174.366,43.423,158.584
C00769=1044.862,406.257,368.713,174.358,43.416,158.582
C00770=1044.852,406.011,368.758,174.349,43.409,158.579
C00771=1044.837,405.601,368.833,174.334,43.398,158.575
C00772=1044.821,405.190,368.907,174.319,43.387,158.571
C00773=1044.805,404.780,368.982,174.304,43.376,158.567
C00774=1044.790,404.369,369.058,174.290,43.365,158.563
C00775=1044.780,404.124,369.102,174.281,43.359,158.561
C00776=1044.772,403.877,369.147,174.272,43.352,158.558
C00777=1044.762,403.632,369.192,174.264,43.346,158.556
C00778=1044.753,403.386,369.236,174.255,43.339,158.553
C00779=1044.743,403.140,369.281,174.246,43.333,158.551
C00780=1044.734,402.894,369.326,174.238,43.326,158.549
C00781=1044.725,402.648,369.369,174.229,43.320,158.546
C00782=1044.716,402.403,369.414,174.220,43.314,158.544
C00783=1044.706,402.157,369.458,174.212,43.307,158.542
C00784=1044.698,401.910,369.503,174.203,43.301,158.539
C00785=1044.688,401.665,369.547,174.195,43.295,158.537
C00786=1044.679,401.419,369.591,174.186,43.288,158.535
C00787=1044.670,401.173,369.636,174.178,43.282,158.532
C00788=1044.660,400.927,369.680,174.169,43.276,158.530
C00789=1044.651,400.681,369.723,174.161,43.269,158.528
C00790=1044.642,400.435,369.768,174.152,43.263,158.526
C00791=1044.633,400.190,369.811,174.144,43.256,158.523
C00792=1044.624,399.944,369.855,174.135,43.251,158.521
C00793=1044.614,399.698,369.899,174.127,43.244,158.519
C00794=1044.606,399.452,369.943,174.119,43.239,158.517
C00795=1044.596,399.206,369.987,174.111,43.232,158.514
C00796=1044.587,398.961,370.031,174.102,43.226,158.512
C00797=1044.578,398.714,370.075,174.094,43.220,158.510
C00798=1044.569,398.468,370.118,174.085,43.214,158.508
C00799=1044.560,398.222,370.162,174.077,43.208,158.506
C00800=1044.551,397.977,370.206,174.070,43.202,158.503
C00801=1044.542,397.730,370.249,174.061,43.196,158.501
C00802=1044.533,397.485,370.293,174.053,43.190,158.499
C00803=1044.524,397.239,370.337,174.045,43.184,158.497
C00804=1044.515,396.992,370.380,174.036,43.178,158.495
C00805=1044.507,396.747,370.424,174.029,43.172,158.492
C00806=1044.497,396.500,370.467,174.021,43.166,158.490
C00807=1044.489,396.255,370.511,174.012,43.160,158.488
C00808=1044.479,396.009,370.554,174.004,43.153,158.486
C00809=1044.470,395.763,370.598,173.997,43.148,158.484
C00810=1044.462,395.517,370.641,173.988,43.142,158.482
C00811=1044.453,395.271,370.684,173.980,43.136,158.480
C00812=1044.444,395.025,370.728,173.973,43.130,158.478
C00813=1044.434,394.779,370.770,173.965,43.125,158.476
C00814=1044.426,394.533,370.813,173.956,43.119,158.473
C00815=1044.417,394.287,370.856,173.949,43.113,158.471
C00816=1044.408,394.041,370.901,173.941,43.107,158.469
C00817=1044.399,393.795,370.943,173.933,43.101,158.467
C00818=1044.390,393.549,370.986,173.925,43.096,158.465
C00819=1044.382,393.303,371.029,173.917,43.090,158.463
C00820=1044.373,393.057,371.072,173.910,43.084,158.461
C00821=1044.363,392.810,371.115,173.902,43.079,158.459
C00822=1044.355,392.564,371.158,173.894,43.073,158.457
C00823=1044.346,392.318,371.201,173.887,43.067,158.455
C00824=1044.338,392.072,371.244,173.878,43.061,158.453
C00825=1044.329,391.826,371.286,173.871,43.055,158.451
C00826=1044.320,391.580,371.329,173.863,43.050,158.449
C00827=1044.306,391.189,371.397,173.851,43.041,158.446
C00828=1044.292,390.797,371.465,173.839,43.032,158.443
C00829=1044.279,390.406,371.532,173.827,43.024,158.439
C00830=1044.264,390.015,371.600,173.815,43.015,158.436
C00831=1044.256,389.768,371.642,173.808,43.009,158.434
C00832=1044.247,389.522,371.684,173.800,43.004,158.432
C00833=1044.239,389.276,371.727,173.793,42.998,158.430
C00834=1044.230,389.029,371.770,173.785,42.992,158.428
C00835=1044.222,388.784,371.811,173.778,42.987,158.426
C00836=1044.213,388.538,371.854,173.770,42.982,158.425
C00837=1044.204,388.291,371.896,173.763,42.976,158.423
C00838=1044.196,388.045,371.938,173.756,42.971,158.421
C00839=1044.187,387.799,371.981,173.748,42.965,158.419
C00840=1044.178,387.553,372.022,173.741,42.960,158.417
C00841=1044.169,387.306,372.064,173.734,42.955,158.415
C00842=1044.161,387.060,372.106,173.726,42.950,158.413
C00843=1044.152,386.814,372.149,173.719,42.944,158.411
C00844=1044.143,386.568,372.190,173.712,42.939,158.409
C00845=1044.134,386.322,372.232,173.704,42.934,158.408
C00846=1044.126,386.075,372.274,173.697,42.928,158.406
C00847=1044.117,385.829,372.316,173.690,42.924,158.404
C00848=1044.108,385.582,372.358,173.682,42.918,158.402
C00849=1044.101,385.336,372.400,173.675,42.913,158.400
C00850=1044.092,385.090,372.441,173.669,42.908,158.398
C00851=1044.083,384.844,372.483,173.661,42.902,158.396
C00852=1044.075,384.598,372.525,173.654,42.897,158.395
C00853=1044.066,384.351,372.567,173.647,42.892,158.393
C00854=1044.058,384.104,372.608,173.639,42.887,158.391
C00855=1044.049,383.859,372.649,173.632,42.882,158.389
C00856=1044.041,383.612,372.691,173.625,42.877,158.387
C00857=1044.032,383.366,372.733,173.619,42.872,158.386
C00858=1044.024,383.119,372.774,173.611,42.866,158.384
C00859=1044.015,382.873,372.815,173.604,42.861,158.382
C00860=1044.008,382.627,372.857,173.597,42.856,158.380
C00861=1043.999,382.380,372.898,173.591,42.851,158.379
C00862=1043.991,382.134,372.940,173.583,42.846,158.377
C00863=1043.982,381.888,372.981,173.576,42.841,158.375
C00864=1043.975,381.641,373.023,173.569,42.836,158.373
C00865=1043.966,381.395,373.064,173.563,42.831,158.371
C00866=1043.958,381.149,373.105,173.556,42.826,158.370
C00867=1043.949,380.902,373.147,173.548,42.821,158.368
C00868=1043.941,380.656,373.188,173.541,42.816,158.366
C00869=1043.933,380.409,373.230,173.535,42.811,158.364
C00870=1043.924,380.163,373.270,173.528,42.806,158.363
C00871=1043.916,379.916,373.311,173.521,42.801,158.361
C00872=1043.908,379.670,373.353,173.515,42.796,158.359
C00873=1043.900,379.424,373.394,173.507,42.791,158.358
C00874=1043.892,379.177,373.435,173.500,42.786,158.356
C00875=1043.883,378.931,373.476,173.494,42.781,158.354
C00876=1043.875,378.685,373.517,173.487,42.776,158.352
C00877=1043.867,378.438,373.558,173.480,42.772,158.351
C00878=1043.859,378.192,373.598,173.474,42.767,158.349
C00879=1043.850,377.945,373.639,173.467,42.762,158.347
C00880=1043.842,377.698,373.680,173.461,42.758,158.346
C00881=1043.834,377.452,373.721,173.454,42.753,158.344
C00882=1043.825,377.205,373.761,173.447,42.748,158.342
C00883=1043.814,376.848,373.820,173.438,42.741,158.340
C00884=1043.801,376.489,373.879,173.428,42.734,158.338
C00885=1043.789,376.132,373.938,173.418,42.727,158.335
C00886=1043.777,375.775,373.997,173.409,42.720,158.333
C00887=1043.769,375.528,374.038,173.402,42.716,158.331
C00888=1043.761,375.281,374.078,173.396,42.711,158.330
C00889=1043.753,375.034,374.118,173.389,42.706,158.328
C00890=1043.745,374.788,374.159,173.383,42.702,158.326
C00891=1043.737,374.542,374.199,173.376,42.697,158.325
C00892=1043.729,374.294,374.240,173.370,42.692,158.323
C00893=1043.720,374.048,374.280,173.363,42.688,158.322
C00894=1043.712,373.802,374.320,173.357,42.684,158.320
C00895=1043.704,373.555,374.360,173.350,42.679,158.318
C00896=1043.696,373.309,374.401,173.344,42.674,158.317
C00897=1043.688,373.062,374.441,173.337,42.670,158.315
C00898=1043.680,372.816,374.481,173.331,42.665,158.314
C00899=1043.673,372.569,374.521,173.324,42.661,158.312
C00900=1043.665,372.322,374.562,173.318,42.656,158.310
C00901=1043.656,372.076,374.601,173.312,42.651,158.309
C00902=1043.648,371.830,374.642,173.305,42.647,158.307
C00903=1043.640,371.583,374.682,173.299,42.642,158.306
C00904=1043.633,371.336,374.722,173.292,42.638,158.304
C00905=1043.625,371.089,374.762,173.286,42.633,158.303
C00906=1043.617,370.843,374.802,173.281,42.629,158.301
C00907=1043.609,370.596,374.842,173.274,42.624,158.300
C00908=1043.601,370.349,374.882,173.268,42.620,158.298
C00909=1043.592,370.103,374.922,173.261,42.616,158.297
C00910=1043.584,369.856,374.962,173.255,42.611,158.295
C00911=1043.576,369.610,375.001,173.249,42.607,158.294
C00912=1043.568,369.363,375.041,173.242,42.602,158.292
C00913=1043.560,369.116,375.081,173.237,42.598,158.291
C00914=1043.552,368.869,375.120,173.231,42.594,158.289
C00915=1043.544,368.622,375.160,173.224,42.589,158.288
C00916=1043.536,368.376,375.199,173.218,42.585,158.286
C00917=1043.528,368.129,375.239,173.212,42.581,158.285
C00918=1043.520,367.882,375.278,173.205,42.576,158.283
C00919=1043.513,367.636,375.318,173.200,42.572,158.282
C00920=1043.504,367.389,375.357,173.194,42.568,158.280
C00921=1043.497,367.142,375.397,173.187,42.564,158.279
C00922=1043.488,366.895,375.436,173.181,42.559,158.277
C00923=1043.480,366.648,375.476,173.176,42.555,158.276
C00924=1043.473,366.402,375.515,173.169,42.551,158.274
C00925=1043.465,366.156,375.555,173.163,42.547,158.273
C00926=1043.457,365.908,375.593,173.157,42.542,158.271
C00927=1043.449,365.661,375.633,173.151,42.538,158.270
C00928=1043.441,365.415,375.672,173.145,42.534,158.269
C00929=1043.434,365.168,375.711,173.139,42.530,158.267
C00930=1043.425,364.921,375.751,173.133,42.526,158.266
C00931=1043.418,364.674,375.791,173.127,42.521,158.264
C00932=1043.410,364.428,375.829,173.122,42.517,158.263
C00933=1043.402,364.181,375.869,173.115,42.513,158.261
C00934=1043.394,363.934,375.907,173.109,42.509,158.260
C00935=1043.387,363.688,375.947,173.103,42.505,158.259
C00936=1043.379,363.440,375.986,173.098,42.501,158.257
C00937=1043.372,363.194,376.025,173.092,42.497,158.256
C00938=1043.364,362.947,376.064,173.086,42.492,158.254
C00939=1043.353,362.608,376.117,173.078,42.487,158.252
C00940=1043.343,362.271,376.171,173.070,42.481,158.251
C00941=1043.332,361.933,376.224,173.061,42.476,158.249
C00942=1043.321,361.594,376.278,173.054,42.470,158.247
C00943=1043.313,361.347,376.316,173.048,42.466,158.245
C00944=1043.306,361.098,376.355,173.042,42.462,158.244
C00945=1043.297,360.852,376.394,173.036,42.458,158.243
C00946=1043.290,360.605,376.432,173.030,42.454,158.241
C00947=1043.282,360.358,376.471,173.025,42.450,158.240
C00948=1043.275,360.111,376.510,173.019,42.446,158.239
C00949=1043.267,359.864,376.548,173.014,42.443,158.237
C00950=1043.259,359.618,376.587,173.008,42.439,158.236
C00951=1043.251,359.370,376.625,173.002,42.435,158.235
C00952=1043.243,359.124,376.663,172.997,42.431,158.233
C00953=1043.235,358.877,376.702,172.991,42.427,158.232
C00954=1043.228,358.630,376.740,172.985,42.422,158.231
C00955=1043.221,358.383,376.779,172.979,42.419,158.229
C00956=1043.213,358.136,376.818,172.973,42.415,158.228
C00957=1043.205,357.890,376.856,172.968,42.411,158.227
C00958=1043.197,357.642,376.895,172.962,42.408,158.225
C00959=1043.190,357.396,376.933,172.956,42.404,158.224
C00960=1043.182,357.149,376.970,172.951,42.400,158.223
C00961=1043.174,356.901,377.009,172.945,42.396,158.222
C00962=1043.167,356.655,377.048,172.940,42.392,158.220
C00963=1043.159,356.407,377.086,172.934,42.388,158.219
C00964=1043.152,356.160,377.124,172.929,42.385,158.218
C00965=1043.144,355.914,377.162,172.923,42.380,158.216
C00966=1043.135,355.667,377.200,172.917,42.377,158.215
C00967=1043.128,355.420,377.238,172.912,42.373,158.214
C00968=1043.121,355.173,377.276,172.906,42.369,158.213
C00969=1043.113,354.925,377.314,172.901,42.365,158.211
C00970=1043.105,354.679,377.352,172.895,42.362,158.210
C00971=1043.098,354.432,377.390,172.890,42.358,158.209
C00972=1043.090,354.185,377.428,172.884,42.354,158.207
C00973=1043.082,353.938,377.466,172.879,42.351,158.206
C00974=1043.075,353.691,377.504,172.873,42.347,158.205
C00975=1043.068,353.444,377.541,172.869,42.343,158.204
C00976=1043.060,353.197,377.580,172.863,42.340,158.203
C00977=1043.052,352.949,377.618,172.858,42.336,158.201
C00978=1043.045,352.703,377.656,172.852,42.332,158.200
C00979=1043.038,352.456,377.693,172.847,42.329,158.199
C00980=1043.030,352.209,377.731,172.841,42.325,158.198
C00981=1043.023,351.962,377.769,172.836,42.321,158.196
C00982=1043.014,351.715,377.806,172.830,42.318,158.195
C00983=1043.007,351.467,377.844,172.825,42.314,158.194
C00984=1043.000,351.220,377.882,172.819,42.311,158.193
C00985=1042.992,350.974,377.920,172.815,42.307,158.192
C00986=1042.985,350.727,377.957,172.809,42.303,158.190
C00987=1042.978,350.480,377.995,172.804,42.299,158.189
C00988=1042.971,350.232,378.032,172.799,42.296,158.188
C00989=1042.963,349.985,378.070,172.793,42.293,158.187
C00990=1042.955,349.738,378.107,172.788,42.289,158.185
C00991=1042.947,349.491,378.145,172.782,42.286,158.184
C00992=1042.940,349.243,378.182,172.778,42.282,158.183
C00993=1042.933,349.016,378.217,172.773,42.279,158.182
C00994=1042.926,348.789,378.251,172.768,42.275,158.181
C00995=1042.919,348.561,378.285,172.763,42.272,158.180
C00996=1042.913,348.333,378.320,172.759,42.269,158.179
C00997=1042.905,348.106,378.355,172.753,42.266,158.178
C00998=1042.898,347.877,378.388,172.748,42.263,158.177
C00999=1042.892,347.649,378.423,172.744,42.259,158.175
C01000=1042.885,347.422,378.458,172.738,42.256,158.174
C01001=1042.877,347.175,378.495,172.734,42.253,158.173
C01002=1042.870,346.927,378.531,172.729,42.249,158.172
C01003=1042.862,346.680,378.569,172.723,42.246,158.171
C01004=1042.854,346.433,378.606,172.718,42.243,158.170
C01005=1042.847,346.186,378.643,172.714,42.239,158.169
C01006=1042.841,345.939,378.680,172.708,42.236,158.167
C01007=1042.833,345.692,378.717,172.703,42.232,158.166
C01008=1042.826,345.445,378.754,172.697,42.229,158.165
C01009=1042.818,345.198,378.791,172.693,42.225,158.164
C01010=1042.811,344.950,378.828,172.688,42.222,158.163
C01011=1042.803,344.703,378.866,172.682,42.218,158.162
C01012=1042.796,344.456,378.902,172.677,42.216,158.161
C01013=1042.789,344.209,378.939,172.673,42.212,158.160
C01014=1042.781,343.962,378.976,172.667,42.208,158.158
C01015=1042.774,343.715,379.013,172.662,42.205,158.157
C01016=1042.766,343.468,379.050,172.658,42.202,158.156
C01017=1042.759,343.220,379.086,172.652,42.198,158.155
C01018=1042.752,342.973,379.124,172.647,42.195,158.154
C01019=1042.744,342.726,379.160,172.642,42.192,158.153
C01020=1042.737,342.478,379.197,172.637,42.189,158.152
C01021=1042.730,342.232,379.234,172.632,42.185,158.151
C01022=1042.723,341.984,379.270,172.627,42.182,158.150
C01023=1042.715,341.737,379.307,172.622,42.179,158.148
C01024=1042.708,341.490,379.344,172.617,42.176,158.147
C01025=1042.701,341.242,379.380,172.612,42.172,158.146
C01026=1042.693,340.995,379.416,172.607,42.169,158.145
C01027=1042.686,340.748,379.453,172.602,42.165,158.144
C01028=1042.679,340.501,379.490,172.597,42.163,158.143
C01029=1042.671,340.253,379.526,172.593,42.159,158.142
C01030=1042.664,340.006,379.562,172.587,42.156,158.141
C01031=1042.656,339.759,379.598,172.583,42.153,158.140
C01032=1042.649,339.512,379.636,172.578,42.150,158.139
C01033=1042.642,339.265,379.672,172.572,42.146,158.138
C01034=1042.634,339.018,379.708,172.568,42.143,158.137
C01035=1042.627,338.770,379.745,172.563,42.140,158.136
C01036=1042.620,338.522,379.781,172.558,42.137,158.134
C01037=1042.612,338.276,379.817,172.553,42.134,158.133
C01038=1042.606,338.028,379.854,172.548,42.131,158.132
C01039=1042.598,337.781,379.889,172.544,42.128,158.131
C01040=1042.591,337.534,379.926,172.539,42.125,158.130
C01041=1042.583,337.286,379.962,172.534,42.121,158.129
C01042=1042.577,337.039,379.998,172.529,42.118,158.128
C01043=1042.569,336.792,380.034,172.524,42.115,158.127
C01044=1042.561,336.544,380.071,172.520,42.112,158.126
C01045=1042.554,336.298,380.107,172.515,42.109,158.125
C01046=1042.547,336.050,380.143,172.510,42.105,158.124
C01047=1042.541,335.803,380.178,172.505,42.102,158.123
C01048=1042.533,335.555,380.215,172.501,42.099,158.122
C01049=1042.526,335.308,380.251,172.496,42.096,158.121
C01050=1042.518,335.061,380.287,172.491,42.093,158.120
C01051=1042.511,334.814,380.323,172.486,42.090,158.119
C01052=1042.505,334.566,380.359,172.482,42.087,158.118
C01053=1042.494,334.230,380.407,172.475,42.083,158.117
C01054=1042.484,333.894,380.456,172.469,42.079,158.115
C01055=1042.475,333.558,380.505,172.462,42.075,158.114
C01056=1042.465,333.221,380.553,172.456,42.071,158.113
C01057=1042.458,332.975,380.589,172.451,42.068,158.112
C01058=1042.450,332.727,380.625,172.446,42.065,158.111
C01059=1042.443,332.480,380.661,172.442,42.062,158.110
C01060=1042.436,332.232,380.696,172.437,42.059,158.109
C01061=1042.429,331.985,380.732,172.433,42.056,158.108
C01062=1042.422,331.737,380.768,172.429,42.053,158.107
C01063=1042.414,331.490,380.803,172.424,42.050,158.106
C01064=1042.408,331.243,380.839,172.419,42.047,158.105
C01065=1042.400,330.995,380.875,172.414,42.044,158.104
C01066=1042.393,330.748,380.910,172.410,42.041,158.103
C01067=1042.386,330.500,380.945,172.405,42.038,158.102
C01068=1042.379,330.253,380.981,172.401,42.035,158.101
C01069=1042.372,330.006,381.016,172.396,42.033,158.100
C01070=1042.364,329.758,381.053,172.391,42.030,158.099
C01071=1042.358,329.511,381.088,172.387,42.026,158.098
C01072=1042.351,329.264,381.123,172.382,42.023,158.097
C01073=1042.343,329.016,381.158,172.378,42.021,158.096
C01074=1042.336,328.769,381.194,172.373,42.018,158.095
C01075=1042.329,328.522,381.229,172.369,42.015,158.094
C01076=1042.321,328.274,381.264,172.364,42.012,158.093
C01077=1042.314,328.027,381.299,172.360,42.009,158.092
C01078=1042.307,327.779,381.334,172.356,42.007,158.091
C01079=1042.299,327.532,381.369,172.350,42.004,158.090
C01080=1042.292,327.284,381.404,172.346,42.001,158.089
C01081=1042.284,327.037,381.439,172.341,41.998,158.088
C01082=1042.277,326.789,381.474,172.337,41.996,158.088
C01083=1042.271,326.542,381.509,172.332,41.993,158.087
C01084=1042.263,326.295,381.544,172.328,41.990,158.086
C01085=1042.256,326.047,381.579,172.324,41.987,158.085
C01086=1042.248,325.800,381.614,172.319,41.985,158.084
C01087=1042.242,325.552,381.649,172.315,41.982,158.083
C01088=1042.234,325.305,381.683,172.311,41.979,158.082
C01089=1042.227,325.057,381.719,172.306,41.977,158.081
C01090=1042.220,324.810,381.754,172.302,41.974,158.080
C01091=1042.212,324.563,381.789,172.298,41.971,158.079
C01092=1042.206,324.315,381.824,172.292,41.968,158.078
C01093=1042.198,324.067,381.858,172.288,41.965,158.077
C01094=1042.191,323.820,381.893,172.283,41.963,158.077
C01095=1042.184,323.573,381.928,172.279,41.960,158.076
C01096=1042.177,323.325,381.963,172.275,41.957,158.075
C01097=1042.169,323.078,381.997,172.270,41.955,158.074
C01098=1042.163,322.830,382.032,172.266,41.952,158.073
C01099=1042.155,322.582,382.067,172.262,41.949,158.072
C01100=1042.148,322.335,382.102,172.258,41.947,158.071
C01101=1042.141,322.088,382.137,172.253,41.944,158.070
C01102=1042.134,321.840,382.171,172.249,41.941,158.069
C01103=1042.127,321.593,382.206,172.245,41.939,158.069
C01104=1042.120,321.346,382.240,172.240,41.936,158.068
C01105=1042.113,321.098,382.275,172.236,41.933,158.067
C01106=1042.106,320.851,382.309,172.232,41.931,158.066
C01107=1042.099,320.603,382.344,172.228,41.928,158.065
C01108=1042.092,320.356,382.378,172.223,41.925,158.064
C01109=1042.082,320.014,382.426,172.217,41.921,158.063
C01110=1042.073,319.673,382.474,172.211,41.918,158.062
C01111=1042.063,319.332,382.521,172.206,41.914,158.061
C01112=1042.054,318.991,382.569,172.199,41.911,158.059
C01113=1042.046,318.744,382.603,172.195,41.908,158.059
C01114=1042.040,318.496,382.638,172.191,41.905,158.058
C01115=1042.032,318.249,382.672,172.187,41.903,158.057
C01116=1042.026,318.002,382.706,172.183,41.900,158.056
C01117=1042.019,317.755,382.741,172.178,41.898,158.055
C01118=1042.012,317.507,382.775,172.174,41.895,158.054
C01119=1042.005,317.259,382.809,172.170,41.893,158.053
C01120=1041.998,317.012,382.844,172.166,41.889,158.052
C01121=1041.991,316.764,382.878,172.162,41.887,158.052
C01122=1041.985,316.516,382.913,172.157,41.884,158.051
C01123=1041.977,316.269,382.947,172.153,41.882,158.050
C01124=1041.971,316.021,382.982,172.149,41.879,158.049
C01125=1041.964,315.774,383.015,172.145,41.877,158.048
C01126=1041.957,315.527,383.050,172.141,41.874,158.047
C01127=1041.950,315.279,383.084,172.137,41.872,158.047
C01128=1041.943,315.031,383.118,172.132,41.869,158.046
C01129=1041.936,314.783,383.152,172.128,41.867,158.045
C01130=1041.929,314.536,383.187,172.124,41.864,158.044
C01131=1041.923,314.289,383.221,172.120,41.861,158.043
C01132=1041.916,314.041,383.255,172.116,41.859,158.042
C01133=1041.909,313.793,383.289,172.112,41.856,158.041
C01134=1041.902,313.546,383.323,172.108,41.853,158.041
C01135=1041.896,313.298,383.357,172.103,41.851,158.040
C01136=1041.889,313.051,383.392,172.099,41.848,158.039
C01137=1041.882,312.803,383.426,172.095,41.846,158.038
C01138=1041.875,312.556,383.460,172.091,41.843,158.037
C01139=1041.869,312.309,383.493,172.087,41.840,158.036
C01140=1041.861,312.061,383.527,172.084,41.839,158.036
C01141=1041.854,311.813,383.561,172.080,41.836,158.035
C01142=1041.847,311.566,383.595,172.076,41.833,158.034
C01143=1041.840,311.317,383.628,172.071,41.832,158.033
C01144=1041.833,311.070,383.661,172.067,41.829,158.033
C01145=1041.826,310.823,383.695,172.063,41.826,158.032
C01146=1041.819,310.575,383.729,172.059,41.824,158.031
C01147=1041.812,310.327,383.763,172.055,41.822,158.030
C01148=1041.805,310.080,383.795,172.051,41.819,158.029
C01149=1041.798,309.832,383.829,172.047,41.817,158.029
C01150=1041.790,309.585,383.863,172.044,41.815,158.028
C01151=1041.783,309.337,383.896,172.039,41.812,158.027
C01152=1041.777,309.089,383.929,172.035,41.810,158.026
C01153=1041.770,308.842,383.963,172.031,41.808,158.026
C01154=1041.763,308.594,383.997,172.027,41.805,158.025
C01155=1041.756,308.346,384.030,172.023,41.803,158.024
C01156=1041.748,308.099,384.063,172.019,41.801,158.023
C01157=1041.741,307.851,384.097,172.015,41.798,158.022
C01158=1041.735,307.604,384.129,172.011,41.796,158.022
C01159=1041.728,307.356,384.163,172.008,41.793,158.021
C01160=1041.720,307.108,384.197,172.004,41.791,158.020
C01161=1041.714,306.861,384.230,172.000,41.789,158.019
C01162=1041.706,306.614,384.263,171.996,41.786,158.019
C01163=1041.699,306.365,384.296,171.991,41.785,158.018
C01164=1041.693,306.118,384.329,171.987,41.782,158.017
C01165=1041.683,305.782,384.375,171.982,41.779,158.016
C01166=1041.674,305.446,384.419,171.977,41.776,158.015
C01167=1041.664,305.109,384.465,171.971,41.772,158.014
C01168=1041.655,304.773,384.509,171.966,41.769,158.013
C01169=1041.648,304.525,384.543,171.963,41.767,158.012
C01170=1041.642,304.278,384.576,171.959,41.765,158.011
C01171=1041.634,304.030,384.610,171.955,41.763,158.011
C01172=1041.628,303.782,384.642,171.951,41.760,158.010
C01173=1041.621,303.535,384.676,171.947,41.758,158.009
C01174=1041.614,303.287,384.708,171.943,41.755,158.008
C01175=1041.607,303.039,384.742,171.939,41.753,158.008
C01176=1041.600,302.792,384.775,171.935,41.751,158.007
C01177=1041.593,302.544,384.808,171.932,41.749,158.006
C01178=1041.587,302.296,384.841,171.928,41.746,158.005
C01179=1041.580,302.048,384.873,171.924,41.744,158.005
C01180=1041.573,301.801,384.907,171.920,41.742,158.004
C01181=1041.566,301.553,384.940,171.916,41.740,158.003
C01182=1041.560,301.305,384.973,171.912,41.737,158.002
C01183=1041.553,301.058,385.005,171.908,41.735,158.002
C01184=1041.546,300.810,385.039,171.905,41.733,158.001
C01185=1041.539,300.563,385.071,171.901,41.731,158.000
C01186=1041.532,300.315,385.104,171.897,41.729,158.000
C01187=1041.526,300.067,385.137,171.894,41.726,157.999
C01188=1041.520,299.819,385.170,171.890,41.724,157.998
C01189=1041.512,299.572,385.203,171.886,41.721,157.997
C01190=1041.506,299.324,385.236,171.883,41.719,157.997
C01191=1041.499,299.077,385.269,171.879,41.717,157.996
C01192=1041.492,298.829,385.302,171.875,41.715,157.995
C01193=1041.486,298.581,385.335,171.871,41.713,157.994
C01194=1041.478,298.333,385.367,171.867,41.710,157.994
C01195=1041.472,298.085,385.400,171.863,41.708,157.993
C01196=1041.466,297.838,385.433,171.860,41.706,157.992
C01197=1041.460,297.590,385.465,171.857,41.703,157.992
C01198=1041.452,297.342,385.498,171.853,41.701,157.991
C01199=1041.446,297.095,385.531,171.849,41.699,157.990
C01200=1041.439,296.847,385.563,171.845,41.697,157.989
C01201=1041.432,296.599,385.596,171.841,41.695,157.989
C01202=1041.425,296.351,385.629,171.837,41.692,157.988
C01203=1041.419,296.104,385.661,171.834,41.690,157.987
C01204=1041.413,295.856,385.694,171.831,41.688,157.987
C01205=1041.406,295.608,385.727,171.827,41.685,157.986
C01206=1041.399,295.361,385.759,171.823,41.683,157.985
C01207=1041.393,295.112,385.791,171.819,41.681,157.984
C01208=1041.386,294.865,385.823,171.816,41.679,157.984
C01209=1041.379,294.617,385.857,171.812,41.677,157.983
C01210=1041.372,294.370,385.889,171.808,41.675,157.982
C01211=1041.366,294.121,385.921,171.805,41.673,157.982
C01212=1041.358,293.873,385.953,171.802,41.671,157.981
C01213=1041.352,293.626,385.986,171.798,41.669,157.980
C01214=1041.345,293.379,386.018,171.794,41.667,157.980
C01215=1041.338,293.131,386.050,171.790,41.665,157.979
C01216=1041.331,292.882,386.083,171.786,41.663,157.978
C01217=1041.325,292.634,386.114,171.784,41.660,157.977
C01218=1041.318,292.387,386.146,171.780,41.658,157.977
C01219=1041.311,292.140,386.179,171.776,41.656,157.976
C01220=1041.304,291.891,386.211,171.772,41.654,157.975
C01221=1041.295,291.571,386.252,171.767,41.651,157.975
C01222=1041.286,291.252,386.294,171.763,41.649,157.974
C01223=1041.278,290.933,386.334,171.758,41.646,157.973
C01224=1041.269,290.613,386.376,171.754,41.643,157.972
C01225=1041.263,290.364,386.408,171.751,41.641,157.971
C01226=1041.256,290.117,386.441,171.747,41.639,157.971
C01227=1041.249,289.869,386.472,171.743,41.637,157.970
C01228=1041.243,289.621,386.505,171.739,41.635,157.969
C01229=1041.236,289.373,386.536,171.737,41.633,157.969
C01230=1041.229,289.126,386.568,171.733,41.631,157.968
C01231=1041.221,288.878,386.600,171.729,41.629,157.967
C01232=1041.215,288.629,386.632,171.725,41.627,157.967
C01233=1041.208,288.382,386.664,171.722,41.625,157.966
C01234=1041.202,288.134,386.696,171.719,41.623,157.965
C01235=1041.195,287.886,386.727,171.715,41.621,157.965
C01236=1041.188,287.639,386.759,171.711,41.619,157.964
C01237=1041.182,287.391,386.791,171.708,41.616,157.963
C01238=1041.175,287.143,386.823,171.705,41.614,157.963
C01239=1041.168,286.896,386.855,171.701,41.612,157.962
C01240=1041.161,286.647,386.887,171.697,41.610,157.961
C01241=1041.154,286.399,386.918,171.695,41.609,157.961
C01242=1041.147,286.151,386.950,171.691,41.607,157.960
C01243=1041.141,285.903,386.981,171.687,41.605,157.960
C01244=1041.134,285.655,387.012,171.683,41.603,157.959
C01245=1041.127,285.408,387.045,171.681,41.601,157.958
C01246=1041.120,285.160,387.076,171.677,41.599,157.958
C01247=1041.114,284.912,387.107,171.673,41.597,157.957
C01248=1041.107,284.664,387.139,171.670,41.595,157.956
C01249=1041.100,284.416,387.170,171.667,41.593,157.956
C01250=1041.093,284.169,387.202,171.663,41.591,157.955
C01251=1041.087,283.921,387.233,171.659,41.589,157.954
C01252=1041.080,283.673,387.265,171.656,41.587,157.954
C01253=1041.073,283.425,387.296,171.653,41.585,157.953
C01254=1041.066,283.177,387.327,171.649,41.583,157.953
C01255=1041.059,282.928,387.359,171.645,41.581,157.952
C01256=1041.053,282.681,387.390,171.643,41.579,157.951
C01257=1041.046,282.433,387.422,171.639,41.577,157.951
C01258=1041.040,282.185,387.453,171.635,41.575,157.950
C01259=1041.033,281.937,387.485,171.633,41.573,157.949
C01260=1041.026,281.690,387.516,171.629,41.572,157.949
C01261=1041.019,281.442,387.547,171.625,41.570,157.948
C01262=1041.013,281.194,387.579,171.622,41.567,157.948
C01263=1041.006,280.946,387.610,171.619,41.565,157.947
C01264=1040.999,280.698,387.642,171.615,41.563,157.946
C01265=1040.992,280.450,387.673,171.612,41.562,157.946
C01266=1040.986,280.201,387.704,171.609,41.560,157.945
C01267=1040.979,279.954,387.735,171.605,41.558,157.944
C01268=1040.973,279.706,387.767,171.602,41.556,157.944
C01269=1040.966,279.458,387.798,171.599,41.554,157.943
C01270=1040.959,279.210,387.830,171.596,41.552,157.943
C01271=1040.952,278.962,387.861,171.592,41.550,157.942
C01272=1040.947,278.714,387.891,171.588,41.548,157.941
C01273=1040.940,278.466,387.923,171.586,41.546,157.941
C01274=1040.933,278.218,387.954,171.582,41.544,157.940
C01275=1040.926,277.970,387.984,171.578,41.542,157.939
C01276=1040.919,277.722,388.016,171.576,41.541,157.939
C01277=1040.911,277.415,388.054,171.572,41.538,157.938
C01278=1040.902,277.106,388.093,171.567,41.536,157.937
C01279=1040.894,276.798,388.132,171.563,41.534,157.937
C01280=1040.886,276.491,388.170,171.559,41.531,157.936
C01281=1040.880,276.242,388.201,171.556,41.530,157.935
C01282=1040.872,275.995,388.232,171.553,41.527,157.935
C01283=1040.866,275.746,388.262,171.549,41.525,157.934
C01284=1040.859,275.498,388.294,171.546,41.524,157.933
C01285=1040.853,275.250,388.324,171.543,41.522,157.933
C01286=1040.846,275.003,388.355,171.539,41.520,157.932
C01287=1040.839,274.754,388.386,171.537,41.518,157.932
C01288=1040.833,274.506,388.417,171.533,41.516,157.931
C01289=1040.825,274.258,388.447,171.529,41.515,157.931
C01290=1040.819,274.011,388.478,171.526,41.513,157.930
C01291=1040.813,273.762,388.509,171.523,41.511,157.929
C01292=1040.805,273.515,388.540,171.520,41.509,157.929
C01293=1040.799,273.266,388.571,171.516,41.507,157.928
C01294=1040.792,273.018,388.602,171.514,41.505,157.928
C01295=1040.786,272.771,388.632,171.510,41.503,157.927
C01296=1040.779,272.522,388.663,171.508,41.502,157.926
C01297=1040.773,272.275,388.694,171.504,41.500,157.926
C01298=1040.765,272.026,388.724,171.500,41.498,157.925
C01299=1040.760,271.779,388.755,171.498,41.496,157.925
C01300=1040.753,271.531,388.786,171.494,41.494,157.924
C01301=1040.746,271.282,388.816,171.491,41.493,157.923
C01302=1040.739,271.034,388.847,171.488,41.491,157.923
C01303=1040.732,270.787,388.877,171.485,41.489,157.922
C01304=1040.726,270.538,388.908,171.481,41.487,157.922
C01305=1040.719,270.290,388.938,171.479,41.485,157.921
C01306=1040.712,270.042,388.969,171.475,41.483,157.921
C01307=1040.706,269.794,388.999,171.472,41.482,157.920
C01308=1040.699,269.546,389.030,171.469,41.480,157.919
C01309=1040.692,269.298,389.060,171.466,41.478,157.919
C01310=1040.686,269.050,389.090,171.462,41.476,157.918
C01311=1040.679,268.802,389.121,171.460,41.475,157.918
C01312=1040.672,268.554,389.151,171.456,41.472,157.917
C01313=1040.665,268.305,389.181,171.453,41.471,157.917
C01314=1040.659,268.058,389.211,171.450,41.469,157.916
C01315=1040.652,267.810,389.243,171.447,41.467,157.915
C01316=1040.645,267.562,389.273,171.444,41.466,157.915
C01317=1040.639,267.314,389.303,171.441,41.464,157.914
C01318=1040.632,267.066,389.333,171.437,41.462,157.914
C01319=1040.625,266.817,389.363,171.435,41.460,157.913
C01320=1040.619,266.570,389.394,171.431,41.459,157.913
C01321=1040.612,266.321,389.424,171.428,41.457,157.912
C01322=1040.605,266.073,389.454,171.425,41.455,157.912
C01323=1040.599,265.825,389.484,171.422,41.453,157.911
C01324=1040.592,265.577,389.514,171.418,41.451,157.910
C01325=1040.585,265.330,389.544,171.416,41.450,157.910
C01326=1040.579,265.081,389.575,171.412,41.448,157.909
C01327=1040.572,264.832,389.604,171.410,41.446,157.909
C01328=1040.565,264.585,389.634,171.407,41.445,157.908
C01329=1040.559,264.336,389.665,171.403,41.443,157.908
C01330=1040.552,264.089,389.695,171.401,41.441,157.907
C01331=1040.545,263.841,389.725,171.397,41.440,157.907
C01332=1040.539,263.592,389.755,171.394,41.437,157.906
C01333=1040.531,263.289,389.791,171.391,41.435,157.905
C01334=1040.523,262.986,389.829,171.387,41.433,157.905
C01335=1040.515,262.682,389.865,171.383,41.431,157.904
C01336=1040.506,262.378,389.901,171.380,41.429,157.903
C01337=1040.500,262.130,389.932,171.377,41.427,157.903
C01338=1040.493,261.882,389.962,171.373,41.426,157.902
C01339=1040.487,261.635,389.992,171.371,41.424,157.902
C01340=1040.480,261.386,390.021,171.367,41.423,157.901
C01341=1040.472,261.139,390.050,171.364,41.420,157.901
C01342=1040.465,260.891,390.080,171.361,41.419,157.900
C01343=1040.458,260.642,390.110,171.358,41.417,157.900
C01344=1040.452,260.394,390.140,171.355,41.416,157.899
C01345=1040.445,260.145,390.169,171.352,41.414,157.899
C01346=1040.439,259.898,390.199,171.349,41.412,157.898
C01347=1040.432,259.649,390.228,171.346,41.411,157.897
C01348=1040.425,259.401,390.258,171.343,41.409,157.897
C01349=1040.418,259.153,390.288,171.340,41.408,157.896
C01350=1040.411,258.904,390.317,171.337,41.406,157.896
C01351=1040.405,258.657,390.347,171.335,41.404,157.895
C01352=1040.398,258.408,390.377,171.331,41.402,157.895
C01353=1040.391,258.161,390.406,171.328,41.401,157.894
C01354=1040.384,257.912,390.436,171.325,41.399,157.894
C01355=1040.378,257.664,390.466,171.322,41.398,157.893
C01356=1040.370,257.416,390.494,171.320,41.396,157.893
C01357=1040.364,257.168,390.524,171.316,41.394,157.892
C01358=1040.357,256.919,390.553,171.314,41.393,157.892
C01359=1040.350,256.671,390.583,171.310,41.391,157.891
C01360=1040.343,256.423,390.613,171.307,41.390,157.891
C01361=1040.337,256.175,390.642,171.305,41.387,157.890
C01362=1040.330,255.927,390.672,171.301,41.386,157.890
C01363=1040.324,255.679,390.701,171.299,41.384,157.889
C01364=1040.317,255.430,390.730,171.296,41.383,157.889
C01365=1040.310,255.182,390.760,171.292,41.381,157.888
C01366=1040.304,254.934,390.789,171.290,41.380,157.888
C01367=1040.296,254.686,390.818,171.287,41.378,157.887
C01368=1040.290,254.438,390.848,171.284,41.376,157.886
C01369=1040.283,254.189,390.877,171.281,41.375,157.886
C01370=1040.277,253.941,390.906,171.279,41.373,157.885
C01371=1040.270,253.694,390.936,171.275,41.372,157.885
C01372=1040.263,253.445,390.965,171.272,41.369,157.884
C01373=1040.257,253.197,390.994,171.270,41.368,157.884
C01374=1040.250,252.948,391.024,171.266,41.366,157.883
C01375=1040.244,252.700,391.053,171.264,41.365,157.883
C01376=1040.237,252.452,391.082,171.261,41.363,157.882
C01377=1040.230,252.204,391.111,171.259,41.362,157.882
C01378=1040.224,251.955,391.140,171.255,41.360,157.881
C01379=1040.217,251.708,391.170,171.252,41.358,157.881
C01380=1040.210,251.459,391.199,171.250,41.356,157.880
C01381=1040.204,251.211,391.229,171.246,41.355,157.880
C01382=1040.198,250.963,391.258,171.244,41.353,157.879
C01383=1040.191,250.714,391.287,171.241,41.351,157.879
C01384=1040.184,250.467,391.316,171.238,41.350,157.878
C01385=1040.177,250.219,391.345,171.235,41.348,157.878
C01386=1040.170,249.970,391.375,171.232,41.346,157.877
C01387=1040.164,249.722,391.404,171.230,41.345,157.877
C01388=1040.158,249.474,391.433,171.227,41.343,157.876
C01389=1040.149,249.169,391.468,171.223,41.341,157.876
C01390=1040.142,248.864,391.504,171.220,41.339,157.875
C01391=1040.134,248.559,391.540,171.216,41.337,157.874
C01392=1040.125,248.254,391.576,171.213,41.335,157.874
C01393=1040.119,248.006,391.605,171.210,41.333,157.873
C01394=1040.113,247.758,391.634,171.207,41.332,157.873
C01395=1040.107,247.510,391.663,171.204,41.330,157.872
C01396=1040.100,247.261,391.692,171.202,41.328,157.872
C01397=1040.093,247.013,391.721,171.199,41.326,157.871
C01398=1040.087,246.765,391.750,171.196,41.325,157.871
C01399=1040.080,246.517,391.779,171.193,41.323,157.870
C01400=1040.074,246.269,391.808,171.191,41.321,157.869
C01401=1040.067,246.020,391.837,171.188,41.320,157.869
C01402=1040.061,245.772,391.866,171.185,41.318,157.868
C01403=1040.054,245.524,391.895,171.182,41.317,157.868
C01404=1040.048,245.276,391.924,171.179,41.315,157.868
C01405=1040.041,245.028,391.953,171.177,41.313,157.867
C01406=1040.035,244.779,391.982,171.174,41.312,157.867
C01407=1040.028,244.531,392.011,171.172,41.310,157.866
C01408=1040.022,244.282,392.039,171.168,41.308,157.865
C01409=1040.015,244.034,392.067,171.166,41.307,157.865
C01410=1040.008,243.786,392.096,171.163,41.305,157.864
C01411=1040.002,243.537,392.126,171.160,41.303,157.864
C01412=1039.995,243.289,392.153,171.158,41.302,157.863
C01413=1039.989,243.041,392.183,171.154,41.300,157.863
C01414=1039.982,242.793,392.211,171.152,41.299,157.863
C01415=1039.975,242.545,392.240,171.149,41.297,157.862
C01416=1039.969,242.296,392.268,171.147,41.296,157.862
C01417=1039.962,242.048,392.297,171.144,41.294,157.861
C01418=1039.956,241.799,392.326,171.142,41.292,157.861
C01419=1039.949,241.552,392.355,171.138,41.291,157.860
C01420=1039.943,241.303,392.383,171.136,41.289,157.860
C01421=1039.936,241.055,392.411,171.133,41.287,157.859
C01422=1039.929,240.807,392.440,171.130,41.285,157.858
C01423=1039.922,240.558,392.469,171.128,41.284,157.858
C01424=1039.916,240.310,392.498,171.125,41.282,157.858
C01425=1039.909,240.061,392.525,171.122,41.281,157.857
C01426=1039.902,239.813,392.554,171.119,41.280,157.857
C01427=1039.896,239.565,392.582,171.117,41.278,157.856
C01428=1039.889,239.317,392.611,171.114,41.277,157.856
C01429=1039.883,239.068,392.638,171.112,41.275,157.855
C01430=1039.876,238.819,392.668,171.109,41.273,157.855
C01431=1039.869,238.571,392.695,171.107,41.272,157.854
C01432=1039.862,238.323,392.724,171.103,41.270,157.854
C01433=1039.856,238.074,392.752,171.101,41.269,157.853
C01434=1039.849,237.827,392.781,171.098,41.267,157.853
C01435=1039.843,237.578,392.808,171.095,41.266,157.852
C01436=1039.836,237.330,392.837,171.093,41.264,157.852
C01437=1039.830,237.082,392.865,171.090,41.262,157.851
C01438=1039.823,236.834,392.894,171.088,41.261,157.851
C01439=1039.816,236.585,392.921,171.085,41.259,157.850
C01440=1039.809,236.336,392.950,171.082,41.258,157.850
C01441=1039.802,236.088,392.978,171.079,41.256,157.849
C01442=1039.796,235.840,393.006,171.077,41.255,157.849
C01443=1039.789,235.592,393.035,171.074,41.253,157.848
C01444=1039.783,235.343,393.063,171.072,41.251,157.848
C01445=1039.774,235.033,393.098,171.068,41.250,157.848
C01446=1039.765,234.722,393.133,171.065,41.248,157.847
C01447=1039.757,234.411,393.168,171.062,41.246,157.846
C01448=1039.749,234.100,393.203,171.059,41.243,157.846
C01449=1039.743,233.852,393.231,171.056,41.242,157.845
C01450=1039.736,233.604,393.260,171.053,41.240,157.845
C01451=1039.730,233.355,393.288,171.050,41.239,157.844
C01452=1039.723,233.107,393.315,171.048,41.238,157.844
C01453=1039.716,232.859,393.344,171.045,41.236,157.843
C01454=1039.710,232.610,393.372,171.043,41.234,157.843
C01455=1039.703,232.362,393.400,171.040,41.233,157.842
C01456=1039.697,232.114,393.428,171.038,41.231,157.842
C01457=1039.691,231.866,393.455,171.035,41.230,157.841
C01458=1039.684,231.618,393.484,171.033,41.228,157.841
C01459=1039.677,231.370,393.511,171.030,41.226,157.840
C01460=1039.671,231.121,393.540,171.028,41.225,157.840
C01461=1039.664,230.872,393.567,171.025,41.223,157.840
C01462=1039.658,230.624,393.595,171.023,41.222,157.839
C01463=1039.651,230.375,393.623,171.020,41.220,157.839
C01464=1039.644,230.127,393.650,171.018,41.218,157.838
C01465=1039.637,229.879,393.679,171.015,41.217,157.838
C01466=1039.631,229.631,393.707,171.012,41.215,157.837
C01467=1039.624,229.382,393.734,171.010,41.214,157.837
C01468=1039.617,229.134,393.762,171.008,41.213,157.836
C01469=1039.610,228.885,393.790,171.005,41.211,157.836
C01470=1039.604,228.637,393.818,171.002,41.209,157.835
C01471=1039.598,228.388,393.846,171.000,41.208,157.835
C01472=1039.590,228.140,393.873,170.997,41.206,157.834
C01473=1039.584,227.892,393.901,170.995,41.205,157.834
C01474=1039.577,227.643,393.928,170.992,41.203,157.833
C01475=1039.570,227.395,393.956,170.990,41.201,157.833
C01476=1039.564,227.146,393.984,170.987,41.200,157.833
C01477=1039.557,226.898,394.012,170.985,41.199,157.832
C01478=1039.551,226.650,394.039,170.982,41.197,157.832
C01479=1039.545,226.401,394.066,170.979,41.196,157.831
C01480=1039.537,226.153,394.093,170.976,41.194,157.831
C01481=1039.530,225.905,394.121,170.974,41.193,157.830
C01482=1039.524,225.656,394.149,170.972,41.191,157.830
C01483=1039.517,225.408,394.176,170.970,41.190,157.829
C01484=1039.510,225.159,394.204,170.967,41.188,157.829
C01485=1039.504,224.911,394.232,170.965,41.187,157.829
C01486=1039.497,224.662,394.259,170.962,41.185,157.828
C01487=1039.490,224.414,394.286,170.960,41.183,157.828
C01488=1039.484,224.166,394.313,170.957,41.182,157.827
C01489=1039.477,223.917,394.341,170.955,41.180,157.827
C01490=1039.471,223.669,394.369,170.952,41.179,157.826
C01491=1039.464,223.420,394.396,170.950,41.178,157.826
C01492=1039.457,223.171,394.424,170.947,41.176,157.825
C01493=1039.451,222.923,394.451,170.945,41.174,157.825
C01494=1039.444,222.676,394.478,170.942,41.173,157.824
C01495=1039.437,222.427,394.506,170.940,41.171,157.824
C01496=1039.431,222.178,394.533,170.937,41.169,157.823
C01497=1039.424,221.930,394.561,170.935,41.168,157.823
C01498=1039.418,221.681,394.588,170.932,41.167,157.823
C01499=1039.411,221.432,394.615,170.930,41.165,157.822
C01500=1039.404,221.185,394.642,170.927,41.164,157.822
C01501=1039.395,220.866,394.677,170.925,41.161,157.821
C01502=1039.387,220.548,394.712,170.921,41.160,157.821
C01503=1039.379,220.230,394.747,170.918,41.158,157.820
C01504=1039.371,219.912,394.782,170.915,41.156,157.819
C01505=1039.364,219.664,394.810,170.913,41.154,157.819
C01506=1039.358,219.415,394.837,170.911,41.153,157.818
C01507=1039.350,219.167,394.864,170.908,41.151,157.818
C01508=1039.344,218.918,394.891,170.906,41.150,157.818
C01509=1039.337,218.670,394.918,170.903,41.148,157.817
C01510=1039.330,218.422,394.945,170.901,41.146,157.817
C01511=1039.323,218.173,394.972,170.898,41.145,157.816
C01512=1039.317,217.925,394.999,170.896,41.144,157.816
C01513=1039.310,217.676,395.026,170.893,41.142,157.815
C01514=1039.303,217.428,395.053,170.891,41.141,157.815
C01515=1039.297,217.179,395.080,170.888,41.140,157.815
C01516=1039.290,216.930,395.107,170.886,41.138,157.814
C01517=1039.283,216.682,395.134,170.884,41.136,157.814
C01518=1039.277,216.434,395.160,170.882,41.135,157.813
C01519=1039.270,216.185,395.188,170.879,41.133,157.813
C01520=1039.263,215.937,395.215,170.877,41.132,157.812
C01521=1039.256,215.688,395.242,170.874,41.130,157.812
C01522=1039.250,215.440,395.269,170.872,41.129,157.811
C01523=1039.243,215.192,395.296,170.869,41.127,157.811
C01524=1039.237,214.943,395.323,170.867,41.126,157.810
C01525=1039.230,214.695,395.349,170.865,41.124,157.810
C01526=1039.223,214.446,395.377,170.863,41.123,157.810
C01527=1039.216,214.197,395.403,170.860,41.121,157.809
C01528=1039.211,213.949,395.430,170.858,41.120,157.809
C01529=1039.203,213.701,395.457,170.855,41.118,157.808
C01530=1039.197,213.452,395.484,170.853,41.116,157.808
C01531=1039.191,213.204,395.511,170.850,41.115,157.807
C01532=1039.184,212.955,395.538,170.849,41.114,157.807
C01533=1039.177,212.706,395.565,170.846,41.112,157.806
C01534=1039.171,212.458,395.591,170.844,41.110,157.806
C01535=1039.164,212.210,395.619,170.841,41.109,157.806
C01536=1039.157,211.961,395.645,170.839,41.107,157.805
C01537=1039.151,211.713,395.672,170.837,41.105,157.805
C01538=1039.144,211.465,395.699,170.835,41.104,157.804
C01539=1039.137,211.216,395.726,170.832,41.103,157.804
C01540=1039.131,210.967,395.752,170.830,41.101,157.803
C01541=1039.124,210.719,395.778,170.827,41.099,157.803
C01542=1039.117,210.470,395.805,170.825,41.098,157.803
C01543=1039.110,210.222,395.832,170.823,41.097,157.802
C01544=1039.103,209.973,395.859,170.821,41.095,157.802
C01545=1039.098,209.725,395.885,170.818,41.093,157.801
C01546=1039.090,209.476,395.912,170.816,41.092,157.801
C01547=1039.084,209.227,395.939,170.814,41.091,157.800
C01548=1039.078,208.979,395.965,170.812,41.089,157.800
C01549=1039.070,208.731,395.992,170.809,41.087,157.799
C01550=1039.063,208.482,396.018,170.807,41.086,157.799
C01551=1039.057,208.234,396.045,170.805,41.085,157.799
C01552=1039.050,207.985,396.071,170.802,41.083,157.798
C01553=1039.044,207.737,396.097,170.801,41.082,157.798
C01554=1039.037,207.488,396.124,170.798,41.080,157.797
C01555=1039.030,207.239,396.151,170.796,41.078,157.797
C01556=1039.024,206.991,396.177,170.793,41.077,157.796
C01557=1039.015,206.679,396.210,170.790,41.075,157.796
C01558=1039.007,206.367,396.243,170.788,41.073,157.795
C01559=1038.998,206.054,396.276,170.785,41.071,157.795
C01560=1038.990,205.741,396.310,170.782,41.070,157.794
C01561=1038.963,204.691,396.416,170.486,40.966,157.757
C01562=1038.957,204.442,396.441,170.483,40.965,157.757
C01563=1038.951,204.194,396.466,170.480,40.964,157.757
C01564=1038.945,203.944,396.491,170.476,40.964,157.757
C01565=1038.939,203.696,396.516,170.474,40.963,157.756
C01566=1038.933,203.447,396.542,170.471,40.962,157.756
C01567=1038.927,203.198,396.567,170.467,40.961,157.756
C01568=1038.921,202.950,396.592,170.464,40.961,157.755
C01569=1038.915,202.701,396.617,170.461,40.960,157.755
C01570=1038.909,202.452,396.642,170.458,40.959,157.755
C01571=1038.902,202.204,396.667,170.455,40.958,157.754
C01572=1038.896,201.955,396.692,170.452,40.957,157.754
C01573=1038.890,201.706,396.717,170.448,40.957,157.754
C01574=1038.884,201.457,396.742,170.446,40.956,157.753
C01575=1038.878,201.209,396.767,170.443,40.955,157.753
C01576=1038.872,200.961,396.792,170.440,40.954,157.753
C01577=1038.866,200.711,396.817,170.436,40.954,157.752
C01578=1038.859,200.463,396.842,170.434,40.953,157.752
C01579=1038.853,200.214,396.866,170.431,40.952,157.752
C01580=1038.846,199.965,396.891,170.427,40.952,157.752
C01581=1038.840,199.718,396.916,170.424,40.951,157.751
C01582=1038.834,199.469,396.940,170.421,40.951,157.751
C01583=1038.828,199.220,396.965,170.419,40.950,157.751
C01584=1038.822,198.971,396.990,170.415,40.949,157.751
C01585=1038.815,198.722,397.015,170.412,40.949,157.750
C01586=1038.809,198.473,397.039,170.409,40.948,157.750
C01587=1038.803,198.225,397.064,170.405,40.947,157.750
C01588=1038.797,197.976,397.088,170.403,40.947,157.749
C01589=1038.790,197.728,397.113,170.400,40.946,157.749
C01590=1038.784,197.478,397.138,170.397,40.946,157.749
C01591=1038.778,197.230,397.163,170.394,40.946,157.749
C01592=1038.772,196.981,397.187,170.391,40.945,157.748
C01593=1038.765,196.733,397.212,170.388,40.944,157.748
C01594=1038.759,196.484,397.236,170.385,40.943,157.748
C01595=1038.753,196.234,397.261,170.381,40.943,157.748
C01596=1038.746,195.987,397.285,170.379,40.942,157.747
C01597=1038.741,195.738,397.310,170.376,40.942,157.747
C01598=1038.734,195.489,397.335,170.373,40.941,157.747
C01599=1038.728,195.240,397.359,170.369,40.941,157.746
C01600=1038.722,194.992,397.383,170.367,40.940,157.746
C01601=1038.715,194.743,397.408,170.364,40.939,157.746
C01602=1038.710,194.494,397.433,170.361,40.939,157.746
C01603=1038.704,194.245,397.456,170.358,40.938,157.745
C01604=1038.697,193.997,397.482,170.355,40.938,157.745
C01605=1038.691,193.748,397.506,170.352,40.937,157.745
C01606=1038.685,193.499,397.530,170.350,40.936,157.745
C01607=1038.678,193.251,397.555,170.346,40.936,157.744
C01608=1038.673,193.001,397.579,170.343,40.935,157.744
C01609=1038.667,192.753,397.603,170.340,40.935,157.744
C01610=1038.661,192.504,397.628,170.337,40.934,157.743
C01611=1038.654,192.256,397.652,170.334,40.934,157.743
C01612=1038.648,192.007,397.677,170.331,40.933,157.743
C01613=1038.642,191.758,397.701,170.329,40.932,157.743
C01614=1038.636,191.509,397.725,170.326,40.932,157.742
C01615=1038.630,191.261,397.750,170.322,40.931,157.742
C01616=1038.624,191.012,397.774,170.320,40.931,157.742
C01617=1038.618,190.763,397.798,170.317,40.930,157.742
C01618=1038.612,190.514,397.823,170.313,40.930,157.741
C01619=1038.605,190.265,397.847,170.311,40.929,157.741
C01620=1038.600,190.017,397.871,170.308,40.928,157.741
C01621=1038.593,189.768,397.896,170.305,40.928,157.741
C01622=1038.587,189.484,397.923,170.301,40.927,157.740
C01623=1038.580,189.200,397.951,170.298,40.927,157.740
C01624=1038.573,188.915,397.979,170.295,40.926,157.740
C01625=1038.566,188.631,398.006,170.292,40.926,157.739
C01626=1038.559,188.382,398.030,170.289,40.925,157.739
C01627=1038.554,188.134,398.055,170.286,40.924,157.739
C01628=1038.547,187.885,398.079,170.283,40.924,157.739
C01629=1038.542,187.636,398.103,170.280,40.923,157.738
C01630=1038.535,187.387,398.127,170.277,40.923,157.738
C01631=1038.530,187.139,398.151,170.275,40.922,157.738
C01632=1038.523,186.890,398.175,170.272,40.922,157.738
C01633=1038.518,186.641,398.200,170.269,40.921,157.737
C01634=1038.512,186.392,398.224,170.266,40.921,157.737
C01635=1038.506,186.143,398.248,170.263,40.920,157.737
C01636=1038.500,185.894,398.272,170.261,40.920,157.737
C01637=1038.494,185.646,398.296,170.258,40.919,157.736
C01638=1038.488,185.397,398.320,170.254,40.918,157.736
C01639=1038.482,185.148,398.344,170.252,40.918,157.736
C01640=1038.476,184.899,398.368,170.249,40.918,157.736
C01641=1038.470,184.651,398.393,170.247,40.917,157.735
C01642=1038.464,184.402,398.416,170.243,40.916,157.735
C01643=1038.458,184.153,398.440,170.241,40.916,157.735
C01644=1038.452,183.905,398.465,170.238,40.915,157.735
C01645=1038.446,183.656,398.489,170.235,40.915,157.734
C01646=1038.441,183.407,398.513,170.232,40.914,157.734
C01647=1038.434,183.158,398.536,170.229,40.914,157.734
C01648=1038.428,182.909,398.560,170.227,40.914,157.734
C01649=1038.421,182.660,398.584,170.224,40.913,157.734
C01650=1038.415,182.412,398.606,170.221,40.913,157.733
C01651=1038.408,182.163,398.630,170.219,40.913,157.733
C01652=1038.402,181.915,398.654,170.215,40.913,157.733
C01653=1038.396,181.665,398.677,170.212,40.912,157.733
C01654=1038.390,181.417,398.701,170.210,40.912,157.733
C01655=1038.383,181.168,398.725,170.207,40.912,157.732
C01656=1038.378,180.919,398.748,170.204,40.911,157.732
C01657=1038.371,180.670,398.772,170.201,40.911,157.732
C01658=1038.365,180.422,398.796,170.198,40.911,157.732
C01659=1038.359,180.172,398.819,170.196,40.910,157.731
C01660=1038.352,179.924,398.842,170.193,40.910,157.731
C01661=1038.346,179.674,398.865,170.190,40.910,157.731
C01662=1038.339,179.426,398.889,170.187,40.909,157.731
C01663=1038.333,179.177,398.912,170.184,40.909,157.731
C01664=1038.327,178.928,398.936,170.182,40.909,157.730
C01665=1038.321,178.680,398.960,170.179,40.908,157.730
C01666=1038.315,178.430,398.983,170.176,40.908,157.730
C01667=1038.309,178.182,399.007,170.173,40.908,157.730
C01668=1038.302,177.933,399.030,170.170,40.907,157.730
C01669=1038.296,177.685,399.053,170.168,40.907,157.729
C01670=1038.290,177.436,399.076,170.165,40.907,157.729
C01671=1038.283,177.187,399.100,170.163,40.906,157.729
C01672=1038.277,176.938,399.123,170.160,40.906,157.729
C01673=1038.271,176.689,399.147,170.156,40.906,157.729
C01674=1038.265,176.440,399.170,170.154,40.905,157.728
C01675=1038.259,176.192,399.193,170.151,40.905,157.728
C01676=1038.253,175.942,399.217,170.149,40.905,157.728
C01677=1038.246,175.693,399.239,170.146,40.904,157.728
C01678=1038.240,175.445,399.263,170.143,40.904,157.728
C01679=1038.234,175.196,399.286,170.140,40.904,157.727
C01680=1038.228,174.947,399.310,170.138,40.904,157.727
C01681=1038.222,174.698,399.333,170.135,40.904,157.727
C01682=1038.216,174.449,399.356,170.133,40.903,157.727
C01683=1038.210,174.201,399.380,170.130,40.903,157.727
C01684=1038.203,173.952,399.402,170.126,40.903,157.726
C01685=1038.197,173.703,399.426,170.124,40.902,157.726
C01686=1038.191,173.418,399.452,170.121,40.902,157.726
C01687=1038.183,173.134,399.479,170.118,40.902,157.726
C01688=1038.177,172.849,399.505,170.115,40.901,157.726
C01689=1038.169,172.564,399.532,170.111,40.901,157.725
C01690=1038.163,172.315,399.555,170.109,40.901,157.725
C01691=1038.157,172.067,399.578,170.106,40.900,157.725
C01692=1038.151,171.817,399.601,170.104,40.900,157.725
C01693=1038.145,171.569,399.625,170.101,40.900,157.725
C01694=1038.138,171.320,399.647,170.099,40.899,157.724
C01695=1038.133,171.071,399.670,170.095,40.899,157.724
C01696=1038.126,170.822,399.694,170.093,40.899,157.724
C01697=1038.120,170.573,399.717,170.090,40.898,157.724
C01698=1038.115,170.324,399.740,170.088,40.898,157.724
C01699=1038.109,170.076,399.763,170.086,40.898,157.723
C01700=1038.102,169.827,399.786,170.083,40.898,157.723
C01701=1038.096,169.578,399.810,170.080,40.898,157.723
C01702=1038.090,169.329,399.833,170.077,40.897,157.723
C01703=1038.084,169.080,399.855,170.075,40.897,157.723
C01704=1038.079,168.831,399.878,170.072,40.897,157.723
C01705=1038.072,168.583,399.901,170.070,40.896,157.722
C01706=1038.066,168.333,399.924,170.066,40.896,157.722
C01707=1038.060,168.085,399.948,170.064,40.895,157.722
C01708=1038.054,167.836,399.971,170.061,40.895,157.722
C01709=1038.048,167.587,399.994,170.059,40.895,157.721
C01710=1038.043,167.338,400.017,170.056,40.895,157.721
C01711=1038.036,167.090,400.039,170.054,40.895,157.721
C01712=1038.030,166.840,400.062,170.051,40.894,157.721
C01713=1038.024,166.591,400.085,170.048,40.894,157.721
C01714=1038.018,166.342,400.108,170.046,40.894,157.721
C01715=1038.013,166.093,400.131,170.043,40.893,157.720
C01716=1038.006,165.845,400.153,170.041,40.893,157.720
C01717=1038.000,165.596,400.177,170.037,40.893,157.720
C01718=1037.994,165.347,400.200,170.035,40.892,157.720
C01719=1037.989,165.099,400.223,170.033,40.892,157.720
C01720=1037.983,164.850,400.246,170.030,40.892,157.720
C01721=1037.976,164.600,400.269,170.028,40.892,157.719
C01722=1037.970,164.352,400.292,170.025,40.892,157.719
C01723=1037.964,164.103,400.315,170.023,40.891,157.719
C01724=1037.959,163.854,400.337,170.020,40.891,157.719
C01725=1037.952,163.605,400.360,170.017,40.890,157.719
C01726=1037.946,163.356,400.383,170.015,40.890,157.718
C01727=1037.941,163.107,400.406,170.012,40.890,157.718
C01728=1037.935,162.858,400.429,170.010,40.889,157.718
C01729=1037.929,162.610,400.452,170.008,40.890,157.718
C01730=1037.923,162.360,400.473,170.004,40.889,157.718
C01731=1037.917,162.111,400.496,170.002,40.889,157.717
C01732=1037.912,161.863,400.519,169.999,40.889,157.717
C01733=1037.906,161.614,400.542,169.997,40.888,157.717
C01734=1037.899,161.365,400.564,169.995,40.888,157.717
C01735=1037.894,161.116,400.587,169.991,40.888,157.717
C01736=1037.888,160.867,400.610,169.989,40.887,157.716
C01737=1037.882,160.618,400.633,169.987,40.887,157.716
C01738=1037.877,160.369,400.656,169.984,40.887,157.716
C01739=1037.870,160.120,400.678,169.982,40.887,157.716
C01740=1037.865,159.871,400.701,169.979,40.886,157.716
C01741=1037.858,159.623,400.723,169.976,40.886,157.716
C01742=1037.852,159.374,400.746,169.974,40.886,157.716
C01743=1037.846,159.125,400.768,169.971,40.886,157.715
C01744=1037.839,158.875,400.790,169.969,40.886,157.715
C01745=1037.833,158.627,400.813,169.966,40.886,157.715
C01746=1037.827,158.377,400.835,169.964,40.885,157.715
C01747=1037.821,158.129,400.857,169.962,40.885,157.715
C01748=1037.815,157.880,400.880,169.959,40.885,157.715
C01749=1037.809,157.631,400.902,169.956,40.885,157.714
C01750=1037.802,157.346,400.928,169.953,40.885,157.714
C01751=1037.795,157.060,400.953,169.950,40.885,157.714
C01752=1037.788,156.776,400.979,169.947,40.885,157.714
C01753=1037.781,156.490,401.004,169.945,40.884,157.714
C01754=1037.775,156.241,401.027,169.942,40.884,157.713
C01755=1037.769,155.993,401.049,169.940,40.884,157.713
C01756=1037.762,155.743,401.071,169.937,40.884,157.713
C01757=1037.757,155.495,401.094,169.934,40.884,157.713
C01758=1037.751,155.245,401.115,169.932,40.884,157.713
C01759=1037.744,154.997,401.138,169.930,40.883,157.713
C01760=1037.738,154.748,401.161,169.927,40.884,157.713
C01761=1037.732,154.499,401.182,169.925,40.883,157.713
C01762=1037.726,154.250,401.205,169.922,40.883,157.712
C01763=1037.720,154.001,401.227,169.920,40.883,157.712
C01764=1037.714,153.753,401.249,169.917,40.883,157.712
C01765=1037.708,153.503,401.271,169.914,40.883,157.712
C01766=1037.702,153.255,401.293,169.912,40.883,157.712
C01767=1037.696,153.006,401.315,169.910,40.883,157.712
C01768=1037.690,152.757,401.338,169.907,40.883,157.712
C01769=1037.684,152.508,401.359,169.905,40.882,157.711
C01770=1037.678,152.258,401.381,169.902,40.883,157.711
C01771=1037.671,152.010,401.403,169.900,40.882,157.711
C01772=1037.665,151.761,401.425,169.898,40.883,157.711
C01773=1037.659,151.512,401.448,169.894,40.882,157.711
C01774=1037.653,151.262,401.469,169.892,40.882,157.711
C01775=1037.647,151.013,401.491,169.890,40.882,157.711
C01776=1037.640,150.765,401.513,169.887,40.882,157.710
C01777=1037.634,150.515,401.535,169.885,40.882,157.710
C01778=1037.629,150.267,401.558,169.883,40.882,157.710
C01779=1037.623,150.018,401.579,169.880,40.881,157.710
C01780=1037.617,149.769,401.601,169.878,40.882,157.710
C01781=1037.610,149.520,401.623,169.875,40.881,157.710
C01782=1037.604,149.271,401.645,169.872,40.882,157.710
C01783=1037.598,149.022,401.666,169.870,40.881,157.709
C01784=1037.592,148.773,401.689,169.868,40.881,157.709
C01785=1037.586,148.524,401.711,169.865,40.881,157.709
C01786=1037.580,148.275,401.733,169.863,40.881,157.709
C01787=1037.574,148.026,401.754,169.861,40.881,157.709
C01788=1037.568,147.777,401.776,169.858,40.881,157.709
C01789=1037.562,147.528,401.798,169.856,40.881,157.709
C01790=1037.556,147.279,401.820,169.853,40.880,157.708
C01791=1037.549,147.030,401.841,169.850,40.881,157.708
C01792=1037.543,146.781,401.864,169.848,40.880,157.708
C01793=1037.537,146.532,401.885,169.846,40.881,157.708
C01794=1037.531,146.284,401.906,169.843,40.881,157.708
C01795=1037.525,146.034,401.928,169.841,40.881,157.708
C01796=1037.519,145.785,401.950,169.839,40.881,157.708
C01797=1037.513,145.536,401.971,169.836,40.881,157.707
C01798=1037.506,145.287,401.994,169.834,40.881,157.707
C01799=1037.500,145.038,402.015,169.832,40.880,157.707
C01800=1037.495,144.790,402.037,169.828,40.881,157.707
C01801=1037.488,144.540,402.058,169.826,40.880,157.707
C01802=1037.482,144.291,402.080,169.824,40.881,157.707
C01803=1037.475,144.042,402.101,169.821,40.881,157.707
C01804=1037.469,143.793,402.123,169.819,40.880,157.707
C01805=1037.463,143.544,402.144,169.817,40.881,157.707
C01806=1037.457,143.295,402.166,169.815,40.880,157.706
C01807=1037.451,143.047,402.188,169.812,40.881,157.706
C01808=1037.445,142.798,402.209,169.810,40.880,157.706
C01809=1037.439,142.548,402.231,169.808,40.880,157.706
